# B&R Automation Studio project NAEUL004C00R13L518F00 (part 61)

#### InputRef.var - Change By Project
```iecst
(*2019-05-20*)
(**)
(*General*)
VAR
	p_eAct : REFERENCE TO eDOAction;
	p_udiMax : REFERENCE TO UDINT;
END_VAR
(**)
(*Configuration*)
VAR
	p_tyDOSettings : REFERENCE TO tyDigitalOutputSettings;
END_VAR
(**)
VAR
	p_bManual : REFERENCE TO BOOL;
	p_bSafetyRlyRst : REFERENCE TO BOOL;
	p_bTLRed : REFERENCE TO BOOL;
	p_bTLAmber : REFERENCE TO BOOL;
	p_bTLGreen : REFERENCE TO BOOL;
	p_bBuzzer : REFERENCE TO BOOL;
	p_bUSBA : REFERENCE TO BOOL;
	p_bUSBB : REFERENCE TO BOOL;
	p_bOvenInfoSigA : REFERENCE TO BOOL;
	p_bOvenInfoSigB : REFERENCE TO BOOL;
	p_bPusherExtCtrl : REFERENCE TO BOOL;
	p_bStopperUnblkCtrlA : REFERENCE TO BOOL;
	p_bStopperUnblkCtrlB : REFERENCE TO BOOL;
	p_bInletStopperRetCtrl : REFERENCE TO BOOL;
	p_eCustomerReq : REFERENCE TO eCustomer;
	p_bInletStopperExtCtrl : REFERENCE TO BOOL;
	p_bMag1SelClampCtrl : REFERENCE TO BOOL;
	p_bMag2SelClampCtrl : REFERENCE TO BOOL;
	p_bMag3SelClampCtrl : REFERENCE TO BOOL;
	p_bMag1SelUnclampCtrl : REFERENCE TO BOOL;
	p_bMag2SelUnclampCtrl : REFERENCE TO BOOL;
	p_bMag3SelUnclampCtrl : REFERENCE TO BOOL;
	p_bMag1FixedClampCtrl : REFERENCE TO BOOL;
	p_bMag1RemoteClampCtrl : REFERENCE TO BOOL;
	p_bMag2FixedClampCtrl : REFERENCE TO BOOL;
	p_bMag2RemoteClampCtrl : REFERENCE TO BOOL;
	p_bMag3FixedClampCtrl : REFERENCE TO BOOL;
	p_bMag3RemoteClampCtrl : REFERENCE TO BOOL;
	p_bInShutterOpenCtrl : REFERENCE TO BOOL;
	p_bInShutterCloseCtrl : REFERENCE TO BOOL;
	p_bOutShutterOpenCtrl : REFERENCE TO BOOL;
	p_bOutShutterCloseCtrl : REFERENCE TO BOOL;
	p_bMag1ConvMtrIn : REFERENCE TO BOOL;
	p_bMag1ConvMtrOut : REFERENCE TO BOOL;
	p_bMag2ConvMtrIn : REFERENCE TO BOOL;
	p_bMag2ConvMtrOut : REFERENCE TO BOOL;
	p_bMag3ConvMtrIn : REFERENCE TO BOOL;
	p_bMag3ConvMtrOut : REFERENCE TO BOOL;
	p_bPushConvMtrOn : REFERENCE TO BOOL;
	p_bMag1WallEngageCtrl : REFERENCE TO BOOL;
	p_bMag2WallEngageCtrl : REFERENCE TO BOOL;
	p_bMag3WallEngageCtrl : REFERENCE TO BOOL;
	p_bMag1SafetyBarRetCtrl : REFERENCE TO BOOL;
	p_bMag2SafetyBarRetCtrl : REFERENCE TO BOOL;
	p_bMag3SafetyBarRetCtrl : REFERENCE TO BOOL;
	p_bSOTMagError1 : REFERENCE TO BOOL;
	p_bSOTMagSizeLarge1 : REFERENCE TO BOOL;
	p_bSOTMagReady1 : REFERENCE TO BOOL;
	p_bSOTMagAvailable1 : REFERENCE TO BOOL;
	p_bSOTMagError2 : REFERENCE TO BOOL;
	p_bSOTMagSizeLarge2 : REFERENCE TO BOOL;
	p_bSOTMagReady2 : REFERENCE TO BOOL;
	p_bSOTMagAvailable2 : REFERENCE TO BOOL;
	p_bSOTMagError3 : REFERENCE TO BOOL;
	p_bSOTMagSizeLarge3 : REFERENCE TO BOOL;
	p_bSOTMagReady3 : REFERENCE TO BOOL;
	p_bSOTMagAvailable3 : REFERENCE TO BOOL;
	p_bSOTMagError4 : REFERENCE TO BOOL;
	p_bSOTMagSizeLarge4 : REFERENCE TO BOOL;
	p_bSOTMagReady4 : REFERENCE TO BOOL;
	p_bSOTMagAvailable4 : REFERENCE TO BOOL;
	p_bMagAWOpenLimByp1 : REFERENCE TO BOOL;
	p_bMagAWOpenLimByp2 : REFERENCE TO BOOL;
	p_bMagAWOpenLimByp3 : REFERENCE TO BOOL;
	p_bMagAWOpenLimByp4 : REFERENCE TO BOOL;
	p_bMagAWSmallLimSen1 : REFERENCE TO BOOL;
	p_bMagAWSmallLimSen2 : REFERENCE TO BOOL;
	p_bMagAWSmallLimSen3 : REFERENCE TO BOOL;
	p_bMagAWSmallLimSen4 : REFERENCE TO BOOL;
END_VAR
(**)
VAR
	p_bRequestToBring1 : REFERENCE TO BOOL;
	p_bRequestToBring2 : REFERENCE TO BOOL;
	p_bRequestToBring3 : REFERENCE TO BOOL;
	p_bRequestToBring4 : REFERENCE TO BOOL;
	p_bRequestToGet1 : REFERENCE TO BOOL;
	p_bRequestToGet2 : REFERENCE TO BOOL;
	p_bRequestToGet3 : REFERENCE TO BOOL;
	p_bRequestToGet4 : REFERENCE TO BOOL;
END_VAR
(**)
VAR
	p_bEntTopStprUnblkCtrl : REFERENCE TO BOOL;
	p_bMidTopStprUnblkCtrl : REFERENCE TO BOOL;
	p_bExtTopStprUnblkCtrl : REFERENCE TO BOOL;
	p_bMidBtmStprUnblkCtrl : REFERENCE TO BOOL;
	p_bExtBtmStprUnblkCtrl : REFERENCE TO BOOL;
	p_bEntTopStprUnblkCtrl2 : REFERENCE TO BOOL;
	p_bMidTopStprUnblkCtrl2 : REFERENCE TO BOOL;
	p_bExtTopStprUnblkCtrl2 : REFERENCE TO BOOL;
	p_bMidBtmStprUnblkCtrl2 : REFERENCE TO BOOL;
	p_bExtBtmStprUnblkCtrl2 : REFERENCE TO BOOL;
	p_bInMagConvMtrOn : REFERENCE TO BOOL;
	p_bOutMagConvMtrOn : REFERENCE TO BOOL;
	p_bInMagConv2MtrOn : REFERENCE TO BOOL;
	p_bOutMagConv2MtrOn : REFERENCE TO BOOL;
	p_bMtrPwrRly : REFERENCE TO BOOL;
END_VAR
(**)
VAR
	p_bMag1FixedClampOpenCtrl : REFERENCE TO BOOL;
	p_bMag1RemoteClampOpenCtrl : REFERENCE TO BOOL;
	p_bMag2FixedClampOpenCtrl : REFERENCE TO BOOL;
	p_bMag2RemoteClampOpenCtrl : REFERENCE TO BOOL;
	p_bMag3FixedClampOpenCtrl : REFERENCE TO BOOL;
	p_bMag3RemoteClampOpenCtrl : REFERENCE TO BOOL;
END_VAR
(**)
VAR
	p_bOutShutterOpenCtrl3 : REFERENCE TO BOOL;
	p_bOutShutterCloseCtrl3 : REFERENCE TO BOOL;
	p_bOutShutterOpenCtrl2 : REFERENCE TO BOOL;
	p_bOutShutterCloseCtrl2 : REFERENCE TO BOOL;
END_VAR
(**)
VAR
	p_bMtrPshrExt : REFERENCE TO BOOL;
	p_bMtrPshrRet : REFERENCE TO BOOL;
	p_bMtrPshrOn : REFERENCE TO BOOL;
	p_bMtrPshrBrakeRls : REFERENCE TO BOOL;
	p_bMtrPshrSpdBinBit0 : REFERENCE TO BOOL;
	p_bMtrPshrSpdBinBit1 : REFERENCE TO BOOL;
	p_bMtrPshrSpdBinBit2 : REFERENCE TO BOOL;
	p_bMtrPshrAlmRst : REFERENCE TO BOOL;
	p_bBypCurtainPBLED : REFERENCE TO BOOL;
	p_bBypCurtainSen : REFERENCE TO BOOL;
	p_bRstCurtainSen : REFERENCE TO BOOL;
END_VAR
(**)
VAR
	p_bScanTrigSig : REFERENCE TO BOOL;
	p_bMag1ExitPCB : REFERENCE TO BOOL;
	p_bMag2ExitPCB : REFERENCE TO BOOL;
	p_bMag3ExitPCB : REFERENCE TO BOOL;
END_VAR
```

### Hermes.typ - Do Not Change!!!
```iecst
(*2021-08-01*)

TYPE
	tyHermesBrdAvlDat : 	STRUCT
		a_tyXMLTableDataBrdAvl : ARRAY[0..200]OF tyXMLTableDat;
		iXMLTableDataBrdAvlTtlIdx : INT;
		bNewBrdAvl : BOOL := TRUE;
	END_STRUCT;
	tyHermesSvyParam : 	STRUCT
		tSndAlive : TIME;
		tRcvAlive : TIME;
		uiSvySvstemPort : UINT;
		iLaneID : INT;
		sMachineId : STRING[80];
		sClientAddress : STRING[15];
		uiClientPort : UINT;
		bFeatureCheckAliveResponse : BOOL;
		bFeatureConfiguration : BOOL;
		bFeatureBoardTracking : BOOL;
		bFeatureQueryWorkOrderInfo : BOOL;
		bFeatureSendWorkOrderInfo : BOOL;
		bFeatureReplyWorkOrderInfo : BOOL;
	END_STRUCT;
	tyHermesRmtParam : 	STRUCT
		uiSvrPort : UINT;
	END_STRUCT;
	tyHermesDSParam : 	STRUCT
		tSndAlive : TIME;
		tRcvAlive : TIME;
		sDownstreamInterfaceId : STRING[80]; (*The ID of the transportation interface on the downstream side*)
		uiSvrPort : UINT;
		iLaneID : INT;
		sMachineId : STRING[80] := '';
		sClientAddress : STRING[15] := '';
		uiClientPort : UINT;
		bFeatureCheckAliveResponse : BOOL;
		bFeatureBoardForecast : BOOL;
		bFeatureSendBoardInfo : BOOL;
	END_STRUCT;
	tyHermesUSParam : 	STRUCT
		tSndAlive : TIME;
		tRcvAlive : TIME;
		uiClntPort : UINT;
		iLaneID : INT;
		sMachineId : STRING[80] := '';
		sHostAddress : STRING[15] := '';
		sUpstreamInterfaceId : STRING[80]; (*The ID of the transportation interface on the upstream side*)
		uiHostPort : UINT;
		bFeatureCheckAliveResponse : BOOL;
		bFeatureBoardForecast : BOOL;
		bFeatureQueryBoardInfo : BOOL;
		bCmpTypeId : BOOL;
		bCmpParam : BOOL;
		bOverwrite : BOOL;
	END_STRUCT;
END_TYPE

(**)

TYPE
	tyHermesConfiguration : 	STRUCT
		a_tyUSParam : ARRAY[0..c_diHermesConfigMaxIdx]OF tyHermesUSParam;
		a_tyDSParam : ARRAY[0..c_diHermesConfigMaxIdx]OF tyHermesDSParam;
		tySvyParam : tyHermesSvyParam;
	END_STRUCT;
END_TYPE

(**)
(**)
(*Action*)

TYPE
	eHermesAction :
		(
		HermesActIdle,
		HermesActBGStartRun,
		HermesActBGStopRun,
		HermesActDeleteOldLog,
		HermesActCreateDir,
		HermesActWriteRetain,
		HermesActWriteRetainLane1,
		HermesActWriteRetainLane2,
		HermesActWriteRetainLane3,
		HermesActWriteRetainLane4,
		HermesActWriteRetainSendWO1,
		HermesActWriteRetainSendWO2,
		HermesActWriteRetainSendWO3,
		HermesActReadRetain,
		HermesActReadRetainLane1,
		HermesActReadRetainLane2,
		HermesActReadRetainLane3,
		HermesActReadRetainLane4,
		HermesActReadRetainSendWO1,
		HermesActReadRetainSendWO2,
		HermesActReadRetainSendWO3,
		HermesActWriteConfig,
		HermesActReadConfig
		);
END_TYPE
```

### Hermes.var - Change By Project
```iecst
(*2019-05-04*)
(**)
(*Action & State & Status*)
VAR
	p_HermesStat : UDINT;
	p_HermesStatus : UDINT;
	p_HermesStatTxt : UDINT;
END_VAR
(**)
(*Alarm*)
VAR
	p_HermesAlmData : UDINT;
END_VAR
(**)
(*Output*)
VAR
	p_HermesFileNotFound : UDINT;
	p_HermesConfiguration : UDINT;
	p_HermesConfigurationWr : UDINT;
	p_HermesUSParam1 : UDINT;
	p_HermesUSParam2 : UDINT;
	p_HermesUSParam3 : UDINT;
	p_HermesUSParam4 : UDINT;
	p_HermesDSParam1 : UDINT;
	p_HermesDSParam2 : UDINT;
	p_HermesDSParam3 : UDINT;
	p_HermesDSParam4 : UDINT;
	p_HermesSvyParam : UDINT;
	p_HermesBrdAvlDataTable1stZ : UDINT;
	p_HermesBrdAvlDataTtlIdx1stZ : UDINT;
	p_HermesBrdAvlDataNewBrdAvl1stZ : UDINT;
	p_HermesBrdAvlDataTableLastZ : UDINT;
	p_HermesBrdAvlDataTtlIdxLastZ : UDINT;
	p_HermesBrdAvlDataNewBrdAvlLastZ : UDINT;
END_VAR
```

### Program Logical/Hermes/Hermes (IEC, version 1.00.0) - 1.00.0 - NtHermes v5.00.0 , NtTCP v5.00.0 , NtMessage v5.00.0

#### Init.st - Change By Project
```iecst
(** 2021-08-01 **)
PROGRAM _INIT

	(* Always Change If Project Change *)

	//Pass Address To Global Address For External Use
	//Action, State & Status
	p_HermesStat	:= ADR(eStat);
	p_HermesStatus	:= ADR(eStatus);
	p_HermesStatTxt	:= ADR(sStatTxt);

	//Alarm
	p_HermesAlmData	:= ADR(tyAlmData);

	//Output
	p_HermesFileNotFound	        	:= ADR(bFileNotFound);
	p_HermesConfiguration	        	:= ADR(tyCurrConfiguration);
	p_HermesConfigurationWr	        	:= ADR(tyConfigurationWr);
	p_HermesUSParam1		        	:= ADR(tyCurrConfiguration.a_tyUSParam[0]); //Lane 1
	p_HermesUSParam2	        		:= ADR(tyCurrConfiguration.a_tyUSParam[1]); //Lane 2
	p_HermesUSParam3		         	:= ADR(tyCurrConfiguration.a_tyUSParam[2]); //Lane 3
	p_HermesUSParam4		        	:= ADR(tyCurrConfiguration.a_tyUSParam[3]); //Lane 4
	p_HermesDSParam1		        	:= ADR(tyCurrConfiguration.a_tyDSParam[0]); //Lane 1
	p_HermesDSParam2		        	:= ADR(tyCurrConfiguration.a_tyDSParam[1]); //Lane 2
	p_HermesDSParam3		         	:= ADR(tyCurrConfiguration.a_tyDSParam[2]); //Lane 3
	p_HermesDSParam4		        	:= ADR(tyCurrConfiguration.a_tyDSParam[3]); //Lane 4
	p_HermesSvyParam		        	:= ADR(tyCurrConfiguration.tySvyParam);
	p_HermesBrdAvlDataTable1stZ		    := ADR(a_tyHermesBrdAvlData[1].a_tyXMLTableDataBrdAvl); //Lane 1 First Zone Data, for B.F
	p_HermesBrdAvlDataTtlIdx1stZ    	:= ADR(a_tyHermesBrdAvlData[1].iXMLTableDataBrdAvlTtlIdx);  //Lane 1 First Zone Data, for B.F
	p_HermesBrdAvlDataNewBrdAvl1stZ	    := ADR(a_tyHermesBrdAvlData[1].bNewBrdAvl);  //Lane 1 First Zone Data, for B.F
	p_HermesBrdAvlDataTableLastZ		:= ADR(a_tyHermesBrdAvlData[1].a_tyXMLTableDataBrdAvl); //Lane 1 Last Zone Data,for B.A, adjust array no. accordingly
	p_HermesBrdAvlDataTtlIdxLastZ	    := ADR(a_tyHermesBrdAvlData[1].iXMLTableDataBrdAvlTtlIdx); //Lane 1 Last Zone Data,for B.A, adjust array no. accordingly
	p_HermesBrdAvlDataNewBrdAvlLastZ	:= ADR(a_tyHermesBrdAvlData[1].bNewBrdAvl); //Lane 1 Last Zone Data,for B.A, adjust array no. accordingly

	(* Always Change If Project Change *)
END_PROGRAM
```

#### Act_InitGlobal.st - Change By Project
```iecst
(** 2021-08-01 **)
ACTION Act_InitGlobal:

	(* Always Change If Project Change *)

	//Pass Data To Link
	p_bLinkStartupRun ACCESS p_StartupRun;

	pa_tyLinkXMLTableDataBrdAvl1 ACCESS p_USHermesATableDataBrdAvl; //lane 1 B.A
	p_iLinkXMLTableDataBrdAvlTtlIdx1 ACCESS p_USHermesATableDataBrdAvlTtlIdx; //lane 1 B.A
//	pa_tyLinkXMLTableDataBrdAvl2 ACCESS p_USHermesTableDataBrdAvl2; //lane 2 B.A
//	p_iLinkXMLTableDataBrdAvlTtlIdx2 ACCESS p_USHermesTableDataBrdAvlTtlIdx2; //lane 2 B.A
//	pa_tyLinkXMLTableDataBrdAvl3 ACCESS p_USHermesTableDataBrdAvl3; //lane 3 B.A
//	p_iLinkXMLTableDataBrdAvlTtlIdx3 ACCESS p_USHermesTableDataBrdAvlTtlIdx3; //lane 3 B.A
//	pa_tyLinkXMLTableDataBrdAvl4 ACCESS p_USHermesTableDataBrdAvl4; //lane 4 B.A
//	p_iLinkXMLTableDataBrdAvlTtlIdx4 ACCESS p_USHermesTableDataBrdAvlTtlIdx4; //lane 4 B.A
	p_eLinkTravLifULPosGo ACCESS p_OpsTravLifULPosGo;
	p_bLinkOpsTravLifULInitDone ACCESS p_OpsTravLifULInitDone; //p_OpsInitConvStepInitDone;
//	p_bLinkOpsInitGConv1MidHvBrd ACCESS p_OpsInitConvMidHvBrd;
	p_bLinkOpsTravLifULEntBrd ACCESS p_OpsTravLifULEntBrd;
	p_bLinkOpsTravLifULExitBrd ACCESS p_OpsTravLifULExitBrd;
	p_bLinkConvHvBrd ACCESS p_PshrConvHvBrd; //p_ConvHvBrd

	p_bLinkUSHermesTransporting ACCESS p_USHermesATransporting;
	p_bLinkUSSMEMATransporting ACCESS p_USSMEMAATransporting;
//	p_bLinkOpsGConv1StepEntBrd ACCESS p_OpsTravLifULEntBrd;// p_OpsConvStepEntBrd;
//	p_bLinkOpsInitGConv2StepInitDone ACCESS p_OpsInitGConv2StepInitDone;  //Zone2
//	p_bLinkOpsInitGConv2MidHvBrd ACCESS p_OpsInitGConv2MidHvBrd;  //Zone2
//	p_bLinkOpsInitGConv2EndHvBrd ACCESS p_OpsInitGConv2EndHvBrd;  //Zone2
//	p_bLinkOpsGConv2HvBrd ACCESS p_OpsGConv2HvBrd;  //Zone2
//	p_bLinkOpsGConv2StepEntBrd ACCESS p_OpsGConv2StepEntBrd;  //Zone2
//	p_bLinkUSSMEMA2Transporting ACCESS p_USSMEMA2Transporting;  //Zone2

	//Pass Data To Internal Use
	p_udiRstErr ACCESS p_RstErrReset;
	p_bPrep ACCESS p_NtParamHermesPrep;
	pa_tyUSParam ACCESS p_UIHermesUSParamWr; //HMI US Configure from UI
	//pa_tyDSParam ACCESS p_UIHermesDSParamWr; //HMI DS Configure from UI
	p_tySvyParam ACCESS p_UIHermesSvyParamWr; //HMI Svy Configure from UI
	p_tyRmtSetConfiguration ACCESS p_RmtHermesSetConfiguration; //US,DS SetConfigure from RmtHermes
	p_tySvySetConfiguration ACCESS p_SvyHermesSetConfiguration; //US,DS SetConfigure from SvyHermes
	p_bRmtPrep ACCESS p_NtParamHermesRmtPrep;
	p_bRmtEn ACCESS p_McParamHermesRmtEn;
	p_bSvyPrep ACCESS p_NtParamHermesSvyPrep;
	p_bSvyEn ACCESS p_McParamHermesSvyEn;
	p_sRetainFileName1 ACCESS p_NtParamHermesRetainFileNm; //lane 1
//	p_sRetainFileName2 ACCESS p_NtParamHermesRetainFileNm2; //lane 2, rename to HermesL2.dat
//	p_sRetainFileName3 ACCESS p_NtParamHermesRetainFileNm3; //lane 3, rename to HermesL3.dat
//	p_sRetainFileName4 ACCESS p_NtParamHermesRetainFileNm4; //lane 4, rename to HermesL4.dat
	p_sConfigFileName ACCESS p_NtParamHermesConfigFileNm;
	p_sProgNm ACCESS p_NtParamHermesProgNm;
	p_bNtSettingsLoadDone ACCESS p_StartupNtSettingsLoadDone;
	p_bRmtHermesWriteConfig ACCESS p_RmtHermesWriteConfig;
	p_bSvyHermesWriteConfig ACCESS p_SvyHermesWriteConfig;
	p_bUISaveHMIConfigure ACCESS p_UISaveHMIConfigure;
	p_bUISaveHMISvyConfig ACCESS p_UISaveHMISvyConfig;
	p_sMcId ACCESS p_McParamMcNm;

	p_bRmtFoundIndexUS1 ACCESS p_RmtHermesFoundIndexUS1;
	p_bRmtFoundIndexUS2 ACCESS p_RmtHermesFoundIndexUS2;
	p_bRmtFoundIndexUS3 ACCESS p_RmtHermesFoundIndexUS3;
	p_bRmtFoundIndexUS4 ACCESS p_RmtHermesFoundIndexUS4;
	p_bRmtFoundIndexDS1 ACCESS p_RmtHermesFoundIndexDS1;
	p_bRmtFoundIndexDS2 ACCESS p_RmtHermesFoundIndexDS2;
	p_bRmtFoundIndexDS3 ACCESS p_RmtHermesFoundIndexDS3;
	p_bRmtFoundIndexDS4 ACCESS p_RmtHermesFoundIndexDS4;
	p_udiRmtIndexUS1 ACCESS p_RmtHermesIndexUS1;
	p_udiRmtIndexUS2 ACCESS p_RmtHermesIndexUS2;
	p_udiRmtIndexUS3 ACCESS p_RmtHermesIndexUS3;
	p_udiRmtIndexUS4 ACCESS p_RmtHermesIndexUS4;
	p_udiRmtIndexDS1 ACCESS p_RmtHermesIndexDS1;
	p_udiRmtIndexDS2 ACCESS p_RmtHermesIndexDS2;
	p_udiRmtIndexDS3 ACCESS p_RmtHermesIndexDS3;
	p_udiRmtIndexDS4 ACCESS p_RmtHermesIndexDS4;

	p_bSvyFoundIndexUS1 ACCESS p_SvyHermesFoundIndexUS1;
	p_bSvyFoundIndexUS2 ACCESS p_SvyHermesFoundIndexUS2;
	p_bSvyFoundIndexUS3 ACCESS p_SvyHermesFoundIndexUS3;
	p_bSvyFoundIndexUS4 ACCESS p_SvyHermesFoundIndexUS4;
	p_bSvyFoundIndexDS1 ACCESS p_SvyHermesFoundIndexDS1;
	p_bSvyFoundIndexDS2 ACCESS p_SvyHermesFoundIndexDS2;
	p_bSvyFoundIndexDS3 ACCESS p_SvyHermesFoundIndexDS3;
	p_bSvyFoundIndexDS4 ACCESS p_SvyHermesFoundIndexDS4;
	p_udiSvyIndexUS1 ACCESS p_SvyHermesIndexUS1;
	p_udiSvyIndexUS2 ACCESS p_SvyHermesIndexUS2;
	p_udiSvyIndexUS3 ACCESS p_SvyHermesIndexUS3;
	p_udiSvyIndexUS4 ACCESS p_SvyHermesIndexUS4;
	p_udiSvyIndexDS1 ACCESS p_SvyHermesIndexDS1;
	p_udiSvyIndexDS2 ACCESS p_SvyHermesIndexDS2;
	p_udiSvyIndexDS3 ACCESS p_SvyHermesIndexDS3;
	p_udiSvyIndexDS4 ACCESS p_SvyHermesIndexDS4;

	p_eLinkMcParamUSACommMod ACCESS p_McParamUSCommAMod;
	p_eLinkMcParamUSBCommMod ACCESS p_McParamUSCommBMod;

	p_bLinkDIRightSen ACCESS p_DIConvRgtSen;
	p_bLinkDIClrSen ACCESS p_DIConvClrSen;

	(* Always Change If Project Change *)
END_ACTION
```

#### InputRef_Link.var - Change By Project
```iecst
(*2021-08-01*)
(**)
VAR
	p_bLinkStartupRun : REFERENCE TO BOOL;
END_VAR
(**)
VAR
	p_eLinkMcParamUSACommMod : REFERENCE TO eMcSetCommMod;
	p_eLinkMcParamUSBCommMod : REFERENCE TO eMcSetCommMod;
	pa_tyLinkXMLTableDataBrdAvl1 : REFERENCE TO ARRAY[0..200] OF tyXMLTableDat;
	p_iLinkXMLTableDataBrdAvlTtlIdx1 : REFERENCE TO INT;
	pa_tyLinkXMLTableDataBrdAvl2 : REFERENCE TO ARRAY[0..200] OF tyXMLTableDat;
	p_iLinkXMLTableDataBrdAvlTtlIdx2 : REFERENCE TO INT;
	pa_tyLinkXMLTableDataBrdAvl3 : REFERENCE TO ARRAY[0..200] OF tyXMLTableDat;
	p_iLinkXMLTableDataBrdAvlTtlIdx3 : REFERENCE TO INT;
	pa_tyLinkXMLTableDataBrdAvl4 : REFERENCE TO ARRAY[0..200] OF tyXMLTableDat;
	p_iLinkXMLTableDataBrdAvlTtlIdx4 : REFERENCE TO INT;
END_VAR
(**)
VAR
	tyHermesBrdAvlData : tyHermesBrdAvlDat;
	a_tyHermesBrdAvlData : ARRAY[1..200] OF tyHermesBrdAvlDat; (*Cater Up to 6 Zones*)
END_VAR
(**)
(*Zone 1*)
VAR
	p_eLinkTravLifULPosGo : REFERENCE TO eTravLifULPos;
	p_bLinkOpsTravLifULInitDone : REFERENCE TO BOOL;
	p_bLinkOpsTravLifULEntBrd : REFERENCE TO BOOL;
	p_bLinkOpsTravLifULExitBrd : REFERENCE TO BOOL;
	p_bLinkConvHvBrd : REFERENCE TO BOOL;
	p_bLinkDIRightSen : REFERENCE TO BOOL;
	p_bLinkDIClrSen : REFERENCE TO BOOL;
	p_bLinkOpsInitGConv1MidHvBrd : REFERENCE TO BOOL;
	p_bLinkOpsInitGConv1EndHvBrd : REFERENCE TO BOOL;
	p_bLinkOpsGConv1StepEntBrd : REFERENCE TO BOOL;
	p_bLinkUSHermesTransporting : REFERENCE TO BOOL;
	p_bLinkUSSMEMATransporting : REFERENCE TO BOOL;
END_VAR
(**)
(*Zone 2*)
VAR
	p_bLinkOpsInitGConv2StepInitDone : REFERENCE TO BOOL;
	p_bLinkOpsInitGConv2MidHvBrd : REFERENCE TO BOOL;
	p_bLinkOpsInitGConv2EndHvBrd : REFERENCE TO BOOL;
	p_bLinkOpsGConv2HvBrd : REFERENCE TO BOOL;
	p_bLinkOpsGConv2StepEntBrd : REFERENCE TO BOOL;
	p_bLinkUSSMEMA2Transporting : REFERENCE TO BOOL;
END_VAR
(**)
```

#### Act_LinkAction.st - Change By Project
```iecst
(** 2021-08-01 **)
ACTION Act_LinkAction:

	IF p_bLinkStartupRun = TRUE THEN
		p_eAct ACCESS p_StartupHermesAct;
	ELSIF p_bSvyHermesWriteConfig THEN //Changed
		p_eAct ACCESS p_SvyHermesAct;
	ELSIF p_bRmtHermesWriteConfig THEN
		p_eAct ACCESS p_RmtHermesAct;
	ELSIF p_bUISaveHMIConfigure OR p_bUISaveHMISvyConfig THEN //Change
		p_eAct ACCESS p_UIHermesAct;
	END_IF

END_ACTION
```

#### Act_Link.st - Change By Project
```iecst
(** 2019-05-04 **)
ACTION Act_Link:

	//If not two lane operating at same time no need Lane
	p_udiRetainDataAddr1	:= ADR(a_tyHermesBrdAvlData);
	p_udiRetainDataLen1  	:= SIZEOF(a_tyHermesBrdAvlData);

	IF p_bLinkStartupRun = FALSE THEN

		//Passing Board Available Memory
		//Init Board
		IF EDGEPOS(p_bLinkOpsTravLifULInitDone = TRUE) THEN

			IF p_bLinkConvHvBrd = FALSE THEN
				a_tyHermesBrdAvlData[1].bNewBrdAvl	:= TRUE;

				bHermesWriteRetainLane1	:= TRUE;
			END_IF

		END_IF

		//Enter Board - US1
		IF p_eLinkTravLifULPosGo = TravLifULPosUS1 AND p_bLinkOpsTravLifULEntBrd = TRUE AND EDGEPOS(p_bLinkConvHvBrd = TRUE) THEN

			IF p_eLinkMcParamUSACommMod = McSetCommModHermes THEN

				a_tyHermesBrdAvlData[1].a_tyXMLTableDataBrdAvl		:= pa_tyLinkXMLTableDataBrdAvl1;
				a_tyHermesBrdAvlData[1].iXMLTableDataBrdAvlTtlIdx	:= p_iLinkXMLTableDataBrdAvlTtlIdx1;
				a_tyHermesBrdAvlData[1].bNewBrdAvl					:= FALSE;

				bHermesWriteRetainLane1	:= TRUE;

			ELSE

				a_tyHermesBrdAvlData[1].bNewBrdAvl	:= TRUE;

				bHermesWriteRetainLane1	:= TRUE;

			END_IF

		END_IF

		//Enter Board - US2
		IF p_eLinkTravLifULPosGo = TravLifULPosUS2 AND p_bLinkOpsTravLifULEntBrd = TRUE AND EDGEPOS(p_bLinkConvHvBrd = TRUE) THEN

			IF p_eLinkMcParamUSBCommMod = McSetCommModHermes THEN

				a_tyHermesBrdAvlData[1].a_tyXMLTableDataBrdAvl		:= pa_tyLinkXMLTableDataBrdAvl2;
				a_tyHermesBrdAvlData[1].iXMLTableDataBrdAvlTtlIdx	:= p_iLinkXMLTableDataBrdAvlTtlIdx2;
				a_tyHermesBrdAvlData[1].bNewBrdAvl					:= FALSE;

				bHermesWriteRetain	:= TRUE;

			ELSE

				a_tyHermesBrdAvlData[1].bNewBrdAvl	:= TRUE;

				bHermesWriteRetain	:= TRUE;

			END_IF

		END_IF

		//Exit Board
		IF p_bLinkOpsTravLifULExitBrd = TRUE AND EDGEPOS(p_bLinkConvHvBrd = FALSE  AND EDGENEG(p_bLinkDIRightSen OR p_bLinkDIClrSen )) THEN
			a_tyHermesBrdAvlData[1].bNewBrdAvl	:= TRUE;
			bHermesWriteRetainLane1	:= TRUE;
		END_IF

		//Write Hermes Retain Data
		IF bHermesWriteRetainLane1 = TRUE THEN
			p_eAct	:= HermesActWriteRetainLane1;

			IF (eStat = HermesActWriteRetainLane1) AND (eStatus = Done) THEN
				p_eAct				:= HermesActIdle;
				bHermesWriteRetainLane1	:= FALSE;
			END_IF
		END_IF

	END_IF

END_ACTION
```

#### Cyclic.st - Do Not Change!!!
```iecst
(** 2021-08-01 **)
PROGRAM _CYCLIC

	IF bInitDone = FALSE THEN
		bInitDone	:= TRUE;

		Act_InitLocal;
		Act_InitGlobal;

	ELSIF bInitialDone = FALSE THEN
		IF p_bNtSettingsLoadDone = TRUE THEN
			bInitialDone	:= TRUE;

			Act_Initial;
		END_IF

	ELSE

		Act_RstErr;
		Act_LinkAction;
		Act_Action;
		Act_LinkEn;

		IF (p_bPrep = TRUE) AND (p_bEn = TRUE) AND (p_bDis = FALSE) THEN
			Act_Link;
			Act_Background;
			Act_Main;

		ELSE
			IF eStat <> HermesActIdle THEN
				eStatus	:= Done;
			ELSE
				eStatus	:= Idle;
			END_IF
		END_IF

		Act_Alarm;

	END_IF

END_PROGRAM
```

#### Act_Initial.st - Do Not Change!!!
```iecst
(** 2021-08-01 **)
ACTION Act_Initial:

	//Initial
	sStatTxt	:= a_sStatText[eStat];

	fbDirCreate1.sDevice	:= 'F';
	fbDirCreate1.sDirName	:= 'User';
	fbDirCreate1(bEn := FALSE);

	fbDirCreate2.sDevice	:= 'User';
	fbDirCreate2.sDirName	:= 'Retain';
	fbDirCreate2(bEn := FALSE);

	fbDirCreate3.sDevice	:= 'User';
	fbDirCreate3.sDirName	:= 'Log';
	fbDirCreate3(bEn := FALSE);

	fbDirCreate4.sDevice	:= 'User';
	fbDirCreate4.sDirName	:= 'MachineParameter';
	fbDirCreate4(bEn := FALSE);

	fbFileRead1.sDevice			:= 'McParam';
	fbFileRead1.sFile			:= p_sConfigFileName;
	fbFileRead1.udiOffset		:= 0;
	fbFileRead1.p_Dest			:= ADR(tyCurrConfiguration);
	fbFileRead1.udiLen			:= SIZEOF(tyCurrConfiguration);
	fbFileRead1(bEn := FALSE);

	fbFileWrite1.sDevice		:= 'McParam';
	fbFileWrite1.sFile			:= p_sConfigFileName;
	fbFileWrite1.udiOffset		:= 0;
	fbFileWrite1.p_Src			:= ADR(tyConfigurationWr);
	fbFileWrite1.udiLen			:= SIZEOF(tyConfigurationWr);
	fbFileWrite1.udiOption		:= 0;
	fbFileWrite1(bEn := FALSE);

	fbFileRead2.sDevice			:= 'Retain';
	fbFileRead2.sFile			:= p_sRetainFileName1;
	fbFileRead2.udiOffset		:= 0;
	fbFileRead2(bEn := FALSE);

	fbFileWrite2.sDevice		:= 'Retain';
	fbFileWrite2.sFile			:= p_sRetainFileName1;
	fbFileWrite2.udiOffset		:= 0;
	fbFileWrite2.udiOption		:= 0;
	fbFileWrite2(bEn := FALSE);

	fbFileRead3.sDevice			:= 'Retain';
	fbFileRead3.sFile			:= p_sRetainFileName2;
	fbFileRead3.udiOffset		:= 0;
	fbFileRead3(bEn := FALSE);

	fbFileWrite3.sDevice		:= 'Retain';
	fbFileWrite3.sFile			:= p_sRetainFileName2;
	fbFileWrite3.udiOffset		:= 0;
	fbFileWrite3.udiOption		:= 0;
	fbFileWrite3(bEn := FALSE);

	fbFileRead4.sDevice			:= 'Retain';
	fbFileRead4.sFile			:= p_sRetainFileName3;
	fbFileRead4.udiOffset		:= 0;
	fbFileRead4(bEn := FALSE);

	fbFileWrite4.sDevice		:= 'Retain';
	fbFileWrite4.sFile			:= p_sRetainFileName3;
	fbFileWrite4.udiOffset		:= 0;
	fbFileWrite4.udiOption		:= 0;
	fbFileWrite4(bEn := FALSE);

	fbFileRead5.sDevice			:= 'Retain';
	fbFileRead5.sFile			:= p_sRetainFileName4;
	fbFileRead5.udiOffset		:= 0;
	fbFileRead5(bEn := FALSE);

	fbFileWrite5.sDevice		:= 'Retain';
	fbFileWrite5.sFile			:= p_sRetainFileName4;
	fbFileWrite5.udiOffset		:= 0;
	fbFileWrite5.udiOption		:= 0;
	fbFileWrite5(bEn := FALSE);

END_ACTION
```

#### Act_InitLocal.st - Do Not Change!!!
```iecst
(** 2021-08-01 **)
ACTION Act_InitLocal:

	//Input Reference Link To Local Variable
	p_eAct ACCESS ADR(eAct);
	p_udiRstErr ACCESS ADR(udiRstErr);
	p_bPrep ACCESS ADR(bPrep);
	p_bEn ACCESS ADR(bEn);
	p_bDis ACCESS ADR(bDis);
	pa_tyUSParam ACCESS ADR(a_tyUSParam);
	pa_tyDSParam ACCESS ADR(a_tyDSParam);
	p_tyRmtParam ACCESS ADR(tyRmtParam);
	p_tySvyParam ACCESS ADR(tySvyParam);
	p_tyRmtSetConfiguration ACCESS ADR(tyRmtSetConfiguration);
	p_tySvySetConfiguration ACCESS ADR(tySvySetConfiguration);
	p_bRmtPrep ACCESS ADR(bRmtPrep);
	p_bRmtEn ACCESS ADR(bRmtEn);
	p_bSvyPrep ACCESS ADR(bSvyPrep);
	p_bSvyEn ACCESS ADR(bSvyEn);
	p_sRetainFileName1 ACCESS ADR(sRetainFileName1);
	p_sRetainFileName2 ACCESS ADR(sRetainFileName2);
	p_sRetainFileName3 ACCESS ADR(sRetainFileName3);
	p_sRetainFileName4 ACCESS ADR(sRetainFileName4);
	p_udiRetainDataAddr1 ACCESS ADR(udiRetainDataAddr1);
	p_udiRetainDataLen1 ACCESS ADR(udiRetainDataLen1);
	p_udiRetainDataAddr2 ACCESS ADR(udiRetainDataAddr2);
	p_udiRetainDataLen2 ACCESS ADR(udiRetainDataLen2);
	p_udiRetainDataAddr3 ACCESS ADR(udiRetainDataAddr3);
	p_udiRetainDataLen3 ACCESS ADR(udiRetainDataLen3);
	p_udiRetainDataAddr4 ACCESS ADR(udiRetainDataAddr4);
	p_udiRetainDataLen4 ACCESS ADR(udiRetainDataLen4);
	p_sConfigFileName ACCESS ADR(sConfigFileName);
	p_sProgNm ACCESS ADR(sProgNm);
	p_bNtSettingsLoadDone ACCESS ADR(bNtSettingsLoadDone);
	p_bRmtHermesWriteConfig ACCESS ADR(bRmtHermesWriteConfig);
	p_bSvyHermesWriteConfig ACCESS ADR(bSvyHermesWriteConfig);
	p_bUISaveHMIConfigure ACCESS ADR(bUISaveHMIConfigure);
	p_bUISaveHMISvyConfig ACCESS ADR(bUISaveHMISvyConfig);
	p_sMcId ACCESS ADR(sMcId);

	p_bRmtFoundIndexUS1 ACCESS ADR(bRmtFoundIndexUS1);
	p_bRmtFoundIndexUS2 ACCESS ADR(bRmtFoundIndexUS2);
	p_bRmtFoundIndexUS3 ACCESS ADR(bRmtFoundIndexUS3);
	p_bRmtFoundIndexUS4 ACCESS ADR(bRmtFoundIndexUS4);
	p_bRmtFoundIndexDS1 ACCESS ADR(bRmtFoundIndexDS1);
	p_bRmtFoundIndexDS2 ACCESS ADR(bRmtFoundIndexDS2);
	p_bRmtFoundIndexDS3 ACCESS ADR(bRmtFoundIndexDS3);
	p_bRmtFoundIndexDS4 ACCESS ADR(bRmtFoundIndexDS4);
	p_udiRmtIndexUS1 ACCESS ADR(udiRmtIndexUS1);
	p_udiRmtIndexUS2 ACCESS ADR(udiRmtIndexUS2);
	p_udiRmtIndexUS3 ACCESS ADR(udiRmtIndexUS3);
	p_udiRmtIndexUS4 ACCESS ADR(udiRmtIndexUS4);
	p_udiRmtIndexDS1 ACCESS ADR(udiRmtIndexDS1);
	p_udiRmtIndexDS2 ACCESS ADR(udiRmtIndexDS2);
	p_udiRmtIndexDS3 ACCESS ADR(udiRmtIndexDS3);
	p_udiRmtIndexDS4 ACCESS ADR(udiRmtIndexDS4);

	p_bSvyFoundIndexUS1 ACCESS ADR(bSvyFoundIndexUS1);
	p_bSvyFoundIndexUS2 ACCESS ADR(bSvyFoundIndexUS2);
	p_bSvyFoundIndexUS3 ACCESS ADR(bSvyFoundIndexUS3);
	p_bSvyFoundIndexUS4 ACCESS ADR(bSvyFoundIndexUS4);
	p_bSvyFoundIndexDS1 ACCESS ADR(bSvyFoundIndexDS1);
	p_bSvyFoundIndexDS2 ACCESS ADR(bSvyFoundIndexDS2);
	p_bSvyFoundIndexDS3 ACCESS ADR(bSvyFoundIndexDS3);
	p_bSvyFoundIndexDS4 ACCESS ADR(bSvyFoundIndexDS4);
	p_udiSvyIndexUS1 ACCESS ADR(udiSvyIndexUS1);
	p_udiSvyIndexUS2 ACCESS ADR(udiSvyIndexUS2);
	p_udiSvyIndexUS3 ACCESS ADR(udiSvyIndexUS3);
	p_udiSvyIndexUS4 ACCESS ADR(udiSvyIndexUS4);
	p_udiSvyIndexDS1 ACCESS ADR(udiSvyIndexDS1);
	p_udiSvyIndexDS2 ACCESS ADR(udiSvyIndexDS2);
	p_udiSvyIndexDS3 ACCESS ADR(udiSvyIndexDS3);
	p_udiSvyIndexDS4 ACCESS ADR(udiSvyIndexDS4);

	//Changed
//	p_bSvyPrep ACCESS ADR(bVoid);
//	p_bSvyEn ACCESS ADR(bVoid);
	p_bSvyHermesWriteConfig ACCESS ADR(bSvyHermesWriteConfig);
END_ACTION
```

#### Act_Action.st - Do Not Change!!!
```iecst
(** 2021-08-01 **)
ACTION Act_Action:

	//Reset Error
	IF (eStatus = Error) AND bRstErr THEN
		p_eAct	:= HermesActIdle;
		eStat	:= HermesActIdle;
	END_IF

	//Set p_eAct
	IF eStatus = Idle (*OR eStatus = Busy*) OR eStatus = Done THEN
		eStat	:= p_eAct;
	END_IF

END_ACTION
```

#### Act_Background.st - Do Not Change!!!
```iecst
(** 2021-08-01 **)
ACTION Act_Background:

	//Update Configuration
		//Changed
	IF p_bSvyPrep = TRUE AND p_bSvyEn = TRUE AND p_bSvyHermesWriteConfig THEN

		IF p_bSvyFoundIndexUS1 THEN
			tyConfigurationWr.a_tyUSParam[0].iLaneID		            := p_tySvySetConfiguration.tyData.a_tyUpstreamConfigurations[p_udiSvyIndexUS1].iUpstreamLaneId;
			tyConfigurationWr.a_tyUSParam[0].sHostAddress           	:= p_tySvySetConfiguration.tyData.a_tyUpstreamConfigurations[p_udiSvyIndexUS1].sHostAddress;
			tyConfigurationWr.a_tyUSParam[0].uiHostPort	                := p_tySvySetConfiguration.tyData.a_tyUpstreamConfigurations[p_udiSvyIndexUS1].uiPort;
			tyConfigurationWr.a_tyUSParam[0].sUpstreamInterfaceId   	:= p_tySvySetConfiguration.tyData.a_tyUpstreamConfigurations[p_udiSvyIndexUS1].sUpstreamInterfaceId;
		END_IF

		IF p_bSvyFoundIndexUS2 THEN
			tyConfigurationWr.a_tyUSParam[1].iLaneID		            := p_tySvySetConfiguration.tyData.a_tyUpstreamConfigurations[p_udiSvyIndexUS2].iUpstreamLaneId;
			tyConfigurationWr.a_tyUSParam[1].sHostAddress           	:= p_tySvySetConfiguration.tyData.a_tyUpstreamConfigurations[p_udiSvyIndexUS2].sHostAddress;
			tyConfigurationWr.a_tyUSParam[1].uiHostPort	                := p_tySvySetConfiguration.tyData.a_tyUpstreamConfigurations[p_udiSvyIndexUS2].uiPort;
			tyConfigurationWr.a_tyUSParam[1].sUpstreamInterfaceId   	:= p_tySvySetConfiguration.tyData.a_tyUpstreamConfigurations[p_udiSvyIndexUS2].sUpstreamInterfaceId;
		END_IF

		IF p_bSvyFoundIndexUS3 THEN
			tyConfigurationWr.a_tyUSParam[2].iLaneID		            := p_tySvySetConfiguration.tyData.a_tyUpstreamConfigurations[p_udiSvyIndexUS3].iUpstreamLaneId;
			tyConfigurationWr.a_tyUSParam[2].sHostAddress           	:= p_tySvySetConfiguration.tyData.a_tyUpstreamConfigurations[p_udiSvyIndexUS3].sHostAddress;
			tyConfigurationWr.a_tyUSParam[2].uiHostPort	                := p_tySvySetConfiguration.tyData.a_tyUpstreamConfigurations[p_udiSvyIndexUS3].uiPort;
			tyConfigurationWr.a_tyUSParam[2].sUpstreamInterfaceId   	:= p_tySvySetConfiguration.tyData.a_tyUpstreamConfigurations[p_udiSvyIndexUS3].sUpstreamInterfaceId;
		END_IF

		IF p_bSvyFoundIndexUS4 THEN
			tyConfigurationWr.a_tyUSParam[3].iLaneID		            := p_tySvySetConfiguration.tyData.a_tyUpstreamConfigurations[p_udiSvyIndexUS4].iUpstreamLaneId;
			tyConfigurationWr.a_tyUSParam[3].sHostAddress           	:= p_tySvySetConfiguration.tyData.a_tyUpstreamConfigurations[p_udiSvyIndexUS4].sHostAddress;
			tyConfigurationWr.a_tyUSParam[3].uiHostPort	                := p_tySvySetConfiguration.tyData.a_tyUpstreamConfigurations[p_udiSvyIndexUS4].uiPort;
			tyConfigurationWr.a_tyUSParam[3].sUpstreamInterfaceId   	:= p_tySvySetConfiguration.tyData.a_tyUpstreamConfigurations[p_udiSvyIndexUS4].sUpstreamInterfaceId;
		END_IF

		IF p_bSvyFoundIndexDS1 THEN
			tyConfigurationWr.a_tyDSParam[0].iLaneID	            	:= p_tySvySetConfiguration.tyData.a_tyDownstreamConfigurations[p_udiSvyIndexDS1].iDownstreamLaneId;
			tyConfigurationWr.a_tyDSParam[0].uiSvrPort               	:= p_tySvySetConfiguration.tyData.a_tyDownstreamConfigurations[p_udiSvyIndexDS1].uiPort;
			tyConfigurationWr.a_tyDSParam[0].sDownstreamInterfaceId  	:= p_tySvySetConfiguration.tyData.a_tyDownstreamConfigurations[p_udiSvyIndexDS1].sDownstreamInterfaceId;
		END_IF

		IF p_bSvyFoundIndexDS2 THEN
			tyConfigurationWr.a_tyDSParam[1].iLaneID	            	:= p_tySvySetConfiguration.tyData.a_tyDownstreamConfigurations[p_udiSvyIndexDS2].iDownstreamLaneId;
			tyConfigurationWr.a_tyDSParam[1].uiSvrPort               	:= p_tySvySetConfiguration.tyData.a_tyDownstreamConfigurations[p_udiSvyIndexDS2].uiPort;
			tyConfigurationWr.a_tyDSParam[1].sDownstreamInterfaceId  	:= p_tySvySetConfiguration.tyData.a_tyDownstreamConfigurations[p_udiSvyIndexDS2].sDownstreamInterfaceId;
		END_IF

		IF p_bSvyFoundIndexDS3 THEN
			tyConfigurationWr.a_tyDSParam[2].iLaneID	            	:= p_tySvySetConfiguration.tyData.a_tyDownstreamConfigurations[p_udiSvyIndexDS3].iDownstreamLaneId;
			tyConfigurationWr.a_tyDSParam[2].uiSvrPort               	:= p_tySvySetConfiguration.tyData.a_tyDownstreamConfigurations[p_udiSvyIndexDS3].uiPort;
			tyConfigurationWr.a_tyDSParam[2].sDownstreamInterfaceId  	:= p_tySvySetConfiguration.tyData.a_tyDownstreamConfigurations[p_udiSvyIndexDS3].sDownstreamInterfaceId;
		END_IF

		IF p_bSvyFoundIndexDS4 THEN
			tyConfigurationWr.a_tyDSParam[3].iLaneID	            	:= p_tySvySetConfiguration.tyData.a_tyDownstreamConfigurations[p_udiSvyIndexDS4].iDownstreamLaneId;
			tyConfigurationWr.a_tyDSParam[3].uiSvrPort               	:= p_tySvySetConfiguration.tyData.a_tyDownstreamConfigurations[p_udiSvyIndexDS4].uiPort;
			tyConfigurationWr.a_tyDSParam[3].sDownstreamInterfaceId  	:= p_tySvySetConfiguration.tyData.a_tyDownstreamConfigurations[p_udiSvyIndexDS4].sDownstreamInterfaceId;
		END_IF

		IF p_tySvySetConfiguration.tyAvl.bMachineId = TRUE THEN

			tyConfigurationWr.a_tyUSParam[0].sMachineId		:= p_tySvySetConfiguration.tyData.sMachineId;
			tyConfigurationWr.a_tyDSParam[0].sMachineId		:= p_tySvySetConfiguration.tyData.sMachineId;
			tyConfigurationWr.tySvyParam.sMachineId		    := p_tySvySetConfiguration.tyData.sMachineId;

		END_IF

		IF p_tySvySetConfiguration.tyAvl.bSupervisorySystemPort = TRUE THEN

			tyConfigurationWr.tySvyParam.uiSvySvstemPort	:= p_tySvySetConfiguration.tyData.uiSupervisorySystemPort;

		END_IF

	ELSIF p_bRmtPrep = TRUE AND p_bRmtEn = TRUE AND p_bRmtHermesWriteConfig THEN

		IF p_bRmtFoundIndexUS1 THEN
			tyConfigurationWr.a_tyUSParam[0].iLaneID		            := p_tyRmtSetConfiguration.tyData.a_tyUpstreamConfigurations[p_udiRmtIndexUS1].iUpstreamLaneId;
			tyConfigurationWr.a_tyUSParam[0].sHostAddress           	:= p_tyRmtSetConfiguration.tyData.a_tyUpstreamConfigurations[p_udiRmtIndexUS1].sHostAddress;
			tyConfigurationWr.a_tyUSParam[0].uiHostPort	                := p_tyRmtSetConfiguration.tyData.a_tyUpstreamConfigurations[p_udiRmtIndexUS1].uiPort;
			tyConfigurationWr.a_tyUSParam[0].sUpstreamInterfaceId   	:= p_tyRmtSetConfiguration.tyData.a_tyUpstreamConfigurations[p_udiRmtIndexUS1].sUpstreamInterfaceId;
		END_IF

		IF p_bRmtFoundIndexUS2 THEN
			tyConfigurationWr.a_tyUSParam[1].iLaneID		            := p_tyRmtSetConfiguration.tyData.a_tyUpstreamConfigurations[p_udiRmtIndexUS2].iUpstreamLaneId;
			tyConfigurationWr.a_tyUSParam[1].sHostAddress           	:= p_tyRmtSetConfiguration.tyData.a_tyUpstreamConfigurations[p_udiRmtIndexUS2].sHostAddress;
			tyConfigurationWr.a_tyUSParam[1].uiHostPort	                := p_tyRmtSetConfiguration.tyData.a_tyUpstreamConfigurations[p_udiRmtIndexUS2].uiPort;
			tyConfigurationWr.a_tyUSParam[1].sUpstreamInterfaceId   	:= p_tyRmtSetConfiguration.tyData.a_tyUpstreamConfigurations[p_udiRmtIndexUS2].sUpstreamInterfaceId;
		END_IF

		IF p_bRmtFoundIndexUS3 THEN
			tyConfigurationWr.a_tyUSParam[2].iLaneID		            := p_tyRmtSetConfiguration.tyData.a_tyUpstreamConfigurations[p_udiRmtIndexUS3].iUpstreamLaneId;
			tyConfigurationWr.a_tyUSParam[2].sHostAddress           	:= p_tyRmtSetConfiguration.tyData.a_tyUpstreamConfigurations[p_udiRmtIndexUS3].sHostAddress;
			tyConfigurationWr.a_tyUSParam[2].uiHostPort	                := p_tyRmtSetConfiguration.tyData.a_tyUpstreamConfigurations[p_udiRmtIndexUS3].uiPort;
			tyConfigurationWr.a_tyUSParam[2].sUpstreamInterfaceId   	:= p_tyRmtSetConfiguration.tyData.a_tyUpstreamConfigurations[p_udiRmtIndexUS3].sUpstreamInterfaceId;
		END_IF

		IF p_bRmtFoundIndexUS4 THEN
			tyConfigurationWr.a_tyUSParam[3].iLaneID		            := p_tyRmtSetConfiguration.tyData.a_tyUpstreamConfigurations[p_udiRmtIndexUS4].iUpstreamLaneId;
			tyConfigurationWr.a_tyUSParam[3].sHostAddress           	:= p_tyRmtSetConfiguration.tyData.a_tyUpstreamConfigurations[p_udiRmtIndexUS4].sHostAddress;
			tyConfigurationWr.a_tyUSParam[3].uiHostPort	                := p_tyRmtSetConfiguration.tyData.a_tyUpstreamConfigurations[p_udiRmtIndexUS4].uiPort;
			tyConfigurationWr.a_tyUSParam[3].sUpstreamInterfaceId   	:= p_tyRmtSetConfiguration.tyData.a_tyUpstreamConfigurations[p_udiRmtIndexUS4].sUpstreamInterfaceId;
		END_IF

		IF p_bRmtFoundIndexDS1 THEN
			tyConfigurationWr.a_tyDSParam[0].iLaneID	            	:= p_tyRmtSetConfiguration.tyData.a_tyDownstreamConfigurations[p_udiRmtIndexDS1].iDownstreamLaneId;
			tyConfigurationWr.a_tyDSParam[0].uiSvrPort               	:= p_tyRmtSetConfiguration.tyData.a_tyDownstreamConfigurations[p_udiRmtIndexDS1].uiPort;
			tyConfigurationWr.a_tyDSParam[0].sDownstreamInterfaceId  	:= p_tyRmtSetConfiguration.tyData.a_tyDownstreamConfigurations[p_udiRmtIndexDS1].sDownstreamInterfaceId;
		END_IF

		IF p_bRmtFoundIndexDS2 THEN
			tyConfigurationWr.a_tyDSParam[1].iLaneID	            	:= p_tyRmtSetConfiguration.tyData.a_tyDownstreamConfigurations[p_udiRmtIndexDS2].iDownstreamLaneId;
			tyConfigurationWr.a_tyDSParam[1].uiSvrPort               	:= p_tyRmtSetConfiguration.tyData.a_tyDownstreamConfigurations[p_udiRmtIndexDS2].uiPort;
			tyConfigurationWr.a_tyDSParam[1].sDownstreamInterfaceId  	:= p_tyRmtSetConfiguration.tyData.a_tyDownstreamConfigurations[p_udiRmtIndexDS2].sDownstreamInterfaceId;
		END_IF

		IF p_bRmtFoundIndexDS3 THEN
			tyConfigurationWr.a_tyDSParam[2].iLaneID	            	:= p_tyRmtSetConfiguration.tyData.a_tyDownstreamConfigurations[p_udiRmtIndexDS3].iDownstreamLaneId;
			tyConfigurationWr.a_tyDSParam[2].uiSvrPort               	:= p_tyRmtSetConfiguration.tyData.a_tyDownstreamConfigurations[p_udiRmtIndexDS3].uiPort;
			tyConfigurationWr.a_tyDSParam[2].sDownstreamInterfaceId  	:= p_tyRmtSetConfiguration.tyData.a_tyDownstreamConfigurations[p_udiRmtIndexDS3].sDownstreamInterfaceId;
		END_IF

		IF p_bRmtFoundIndexDS4 THEN
			tyConfigurationWr.a_tyDSParam[3].iLaneID	            	:= p_tyRmtSetConfiguration.tyData.a_tyDownstreamConfigurations[p_udiRmtIndexDS4].iDownstreamLaneId;
			tyConfigurationWr.a_tyDSParam[3].uiSvrPort               	:= p_tyRmtSetConfiguration.tyData.a_tyDownstreamConfigurations[p_udiRmtIndexDS4].uiPort;
			tyConfigurationWr.a_tyDSParam[3].sDownstreamInterfaceId  	:= p_tyRmtSetConfiguration.tyData.a_tyDownstreamConfigurations[p_udiRmtIndexDS4].sDownstreamInterfaceId;
		END_IF

		IF p_tyRmtSetConfiguration.tyAvl.bMachineId = TRUE THEN

			tyConfigurationWr.a_tyUSParam[0].sMachineId		:= p_tyRmtSetConfiguration.tyData.sMachineId;
			tyConfigurationWr.a_tyDSParam[0].sMachineId		:= p_tyRmtSetConfiguration.tyData.sMachineId;
			tyConfigurationWr.tySvyParam.sMachineId		    := p_tyRmtSetConfiguration.tyData.sMachineId;

		END_IF

		IF p_tyRmtSetConfiguration.tyAvl.bSupervisorySystemPort = TRUE THEN

			tyConfigurationWr.tySvyParam.uiSvySvstemPort	:= p_tyRmtSetConfiguration.tyData.uiSupervisorySystemPort;

		END_IF

	ELSIF p_bUISaveHMIConfigure THEN //Save US, DS Configure in HMI

		tyConfigurationWr.a_tyUSParam[0]  := pa_tyUSParam[0]; //lane 1 US
		tyConfigurationWr.a_tyDSParam[0]  := pa_tyDSParam[0]; //lane 1 DS
		tyConfigurationWr.a_tyUSParam[1]  := pa_tyUSParam[1]; //lane 2 US
		tyConfigurationWr.a_tyDSParam[1]  := pa_tyDSParam[1]; //lane 2 DS
		tyConfigurationWr.a_tyUSParam[2]  := pa_tyUSParam[2]; //lane 3 US
		tyConfigurationWr.a_tyDSParam[2]  := pa_tyDSParam[2]; //lane 3 DS
		tyConfigurationWr.a_tyUSParam[3]  := pa_tyUSParam[3]; //lane 4 US
		tyConfigurationWr.a_tyDSParam[3]  := pa_tyDSParam[3]; //lane 4 DS

	ELSIF p_bUISaveHMISvyConfig THEN //Save Supervisory Configure in HMI

		tyConfigurationWr.tySvyParam  := p_tySvyParam;

	END_IF

END_ACTION
```

#### Act_Main.st - Do Not Change!!!
```iecst
(** 2021-08-01 **)
ACTION Act_Main:

	IF eStatOld <> eStat THEN
		fbDirCreate1(bEn := FALSE);
		fbDirCreate2(bEn := FALSE);
		fbDirCreate3(bEn := FALSE);
		fbDirCreate4(bEn := FALSE);
		fbFileRead1(bEn := FALSE);
		fbFileWrite1(bEn := FALSE);
		fbFileRead2(bEn := FALSE);
		fbFileWrite2(bEn := FALSE);
		fbFileRead3(bEn := FALSE);
		fbFileWrite3(bEn := FALSE);
		fbFileRead4(bEn := FALSE);
		fbFileWrite4(bEn := FALSE);
		fbFileRead5(bEn := FALSE);
		fbFileWrite5(bEn := FALSE);
		usiStep			:= 0;
		bFileNotFound	:= FALSE;

		sStatTxt	:= a_sStatText[eStat];

		eStatOld	:= eStat;

		eStatus		:= Busy;
	END_IF

	//Main
	CASE eStat OF

		HermesActIdle:
			eStatus	:= Idle;

		HermesActCreateDir:
			IF eStatus = Idle OR eStatus = Busy THEN

				eStatus	:= Busy;

				CASE usiStep OF
					0:
						fbDirCreate1(bEn := TRUE);
						IF fbDirCreate1.udiStatus = 0 THEN
							usiStep	:= 1;
						ELSIF fbDirCreate1.udiStatus < 65534 THEN
							eStatus		:= Error;

							IF fbDirCreate1.udiStatus = 1908 THEN
								udiStatus	:= 10000;	//Create User Directory Error
							ELSE
								udiStatus	:= fbDirCreate1.udiStatus;
							END_IF
						END_IF

					1:
						fbDirCreate2(bEn := TRUE);
						IF fbDirCreate2.udiStatus = 0 THEN
							usiStep	:= 2;
						ELSIF fbDirCreate2.udiStatus < 65534 THEN
							eStatus		:= Error;

							IF fbDirCreate2.udiStatus = 1908 THEN
								udiStatus	:= 10001;	//Create Retain Directory Error
							ELSE
								udiStatus	:= fbDirCreate2.udiStatus;
							END_IF
						END_IF

					2:
						fbDirCreate3(bEn := TRUE);
						IF fbDirCreate3.udiStatus = 0 THEN
							usiStep	:= 3;
						ELSIF fbDirCreate3.udiStatus < 65534 THEN
							eStatus		:= Error;

							IF fbDirCreate3.udiStatus = 1908 THEN
								udiStatus	:= 10010;	//Create Log Directory Error
							ELSE
								udiStatus	:= fbDirCreate3.udiStatus;
							END_IF
						END_IF

					3:
						fbDirCreate4(bEn := TRUE);
						IF fbDirCreate4.udiStatus = 0 THEN
							eStatus	:= Done;
						ELSIF fbDirCreate4.udiStatus < 65534 THEN
							eStatus		:= Error;

							IF fbDirCreate4.udiStatus = 1908 THEN
								udiStatus	:= 10011;	//Create Machine Parameter Directory Error
							ELSE
								udiStatus	:= fbDirCreate4.udiStatus;
							END_IF
						END_IF

				END_CASE

			END_IF

		HermesActReadRetainLane1:
			IF eStatus = Idle OR eStatus = Busy THEN

				eStatus	:= Busy;

				fbFileRead2.p_Dest	:= p_udiRetainDataAddr1;
				fbFileRead2.udiLen	:= p_udiRetainDataLen1;
				fbFileRead2(bEn := TRUE);

				IF fbFileRead2.udiStatus = 0 THEN
					eStatus	:= Done;
				ELSIF fbFileRead2.udiStatus < 65534 THEN
					eStatus	:= Error;

					IF fbFileRead2.udiStatus = 1900 THEN
						udiStatus	:= 10002;	//File Open Error While Reading Retain File
					ELSIF fbFileRead2.udiStatus = 1902 THEN
						udiStatus	:= 10003;	//File Read Error While Reading Retain File
					ELSIF fbFileRead2.udiStatus = 1904 THEN
						udiStatus	:= 10004;	//File Close Error While Reading Retain File
					ELSIF fbFileRead2.udiStatus = 1915 THEN
						eStatus			:= Done;
						bFileNotFound	:= TRUE;
					ELSE
						udiStatus	:= fbFileRead2.udiStatus;
					END_IF
				END_IF

			END_IF

		HermesActWriteRetainLane1:
			IF eStatus = Idle OR eStatus = Busy THEN

				eStatus	:= Busy;

				fbFileWrite2.p_Src	:= p_udiRetainDataAddr1;
				fbFileWrite2.udiLen	:= p_udiRetainDataLen1;
				fbFileWrite2(bEn := TRUE);

				IF fbFileWrite2.udiStatus = 0 THEN
					eStatus	:= Done;
				ELSIF fbFileWrite2.udiStatus < 65534 THEN
					eStatus	:= Error;

					IF fbFileWrite2.udiStatus = 1900 THEN
						udiStatus	:= 10005;	//File Open Error While Writing Retain File
					ELSIF fbFileWrite2.udiStatus = 1901 THEN
						udiStatus	:= 10006;	//File Create Error While Writing Retain File
					ELSIF fbFileWrite2.udiStatus = 1903 THEN
						udiStatus	:= 10007;	//File Write Error While Writing Retain File
					ELSIF fbFileWrite2.udiStatus = 1904 THEN
						udiStatus	:= 10008;	//File Close Error While Writing Retain File
					ELSIF fbFileWrite2.udiStatus = 1914 THEN
						udiStatus	:= 10009;	//Directory Does Not Exist While Writing Retain File
					ELSE
						udiStatus	:= fbFileWrite2.udiStatus;
					END_IF
				END_IF

			END_IF

		HermesActReadRetainLane2:
			IF eStatus = Idle OR eStatus = Busy THEN

				eStatus	:= Busy;

				fbFileRead3.p_Dest	:= p_udiRetainDataAddr2;
				fbFileRead3.udiLen	:= p_udiRetainDataLen2;
				fbFileRead3(bEn := TRUE);

				IF fbFileRead3.udiStatus = 0 THEN
					eStatus	:= Done;
				ELSIF fbFileRead3.udiStatus < 65534 THEN
					eStatus	:= Error;

					IF fbFileRead3.udiStatus = 1900 THEN
						udiStatus	:= 10032;	//File Open Error While Reading Retain File
					ELSIF fbFileRead3.udiStatus = 1902 THEN
						udiStatus	:= 10033;	//File Read Error While Reading Retain File
					ELSIF fbFileRead3.udiStatus = 1904 THEN
						udiStatus	:= 10034;	//File Close Error While Reading Retain File
					ELSIF fbFileRead3.udiStatus = 1915 THEN
						eStatus			:= Done;
						bFileNotFound	:= TRUE;
					ELSE
						udiStatus	:= fbFileRead3.udiStatus;
					END_IF
				END_IF

			END_IF

		HermesActWriteRetainLane2:
			IF eStatus = Idle OR eStatus = Busy THEN

				eStatus	:= Busy;

				fbFileWrite3.p_Src	:= p_udiRetainDataAddr2;
				fbFileWrite3.udiLen	:= p_udiRetainDataLen2;
				fbFileWrite3(bEn := TRUE);

				IF fbFileWrite3.udiStatus = 0 THEN
					eStatus	:= Done;
				ELSIF fbFileWrite3.udiStatus < 65534 THEN
					eStatus	:= Error;

					IF fbFileWrite3.udiStatus = 1900 THEN
						udiStatus	:= 10035;	//File Open Error While Writing Retain File
					ELSIF fbFileWrite3.udiStatus = 1901 THEN
						udiStatus	:= 10036;	//File Create Error While Writing Retain File
					ELSIF fbFileWrite3.udiStatus = 1903 THEN
						udiStatus	:= 10037;	//File Write Error While Writing Retain File
					ELSIF fbFileWrite3.udiStatus = 1904 THEN
						udiStatus	:= 10038;	//File Close Error While Writing Retain File
					ELSIF fbFileWrite3.udiStatus = 1914 THEN
						udiStatus	:= 10039;	//Directory Does Not Exist While Writing Retain File
					ELSE
						udiStatus	:= fbFileWrite3.udiStatus;
					END_IF
				END_IF

			END_IF

		HermesActReadRetainLane3:
			IF eStatus = Idle OR eStatus = Busy THEN

				eStatus	:= Busy;

				fbFileRead4.p_Dest	:= p_udiRetainDataAddr3;
				fbFileRead4.udiLen	:= p_udiRetainDataLen3;
				fbFileRead4(bEn := TRUE);

				IF fbFileRead4.udiStatus = 0 THEN
					eStatus	:= Done;
				ELSIF fbFileRead4.udiStatus < 65534 THEN
					eStatus	:= Error;

					IF fbFileRead4.udiStatus = 1900 THEN
						udiStatus	:= 10042;	//File Open Error While Reading Retain File
					ELSIF fbFileRead4.udiStatus = 1902 THEN
						udiStatus	:= 10043;	//File Read Error While Reading Retain File
					ELSIF fbFileRead4.udiStatus = 1904 THEN
						udiStatus	:= 10044;	//File Close Error While Reading Retain File
					ELSIF fbFileRead4.udiStatus = 1915 THEN
						eStatus			:= Done;
						bFileNotFound	:= TRUE;
					ELSE
						udiStatus	:= fbFileRead4.udiStatus;
					END_IF
				END_IF

			END_IF

		HermesActWriteRetainLane3:
			IF eStatus = Idle OR eStatus = Busy THEN

				eStatus	:= Busy;

				fbFileWrite4.p_Src	:= p_udiRetainDataAddr3;
				fbFileWrite4.udiLen	:= p_udiRetainDataLen3;
				fbFileWrite4(bEn := TRUE);

				IF fbFileWrite4.udiStatus = 0 THEN
					eStatus	:= Done;
				ELSIF fbFileWrite4.udiStatus < 65534 THEN
					eStatus	:= Error;

					IF fbFileWrite4.udiStatus = 1900 THEN
						udiStatus	:= 10045;	//File Open Error While Writing Retain File
					ELSIF fbFileWrite4.udiStatus = 1901 THEN
						udiStatus	:= 10046;	//File Create Error While Writing Retain File
					ELSIF fbFileWrite4.udiStatus = 1903 THEN
						udiStatus	:= 10047;	//File Write Error While Writing Retain File
					ELSIF fbFileWrite4.udiStatus = 1904 THEN
						udiStatus	:= 10048;	//File Close Error While Writing Retain File
					ELSIF fbFileWrite4.udiStatus = 1914 THEN
						udiStatus	:= 10049;	//Directory Does Not Exist While Writing Retain File
					ELSE
						udiStatus	:= fbFileWrite4.udiStatus;
					END_IF
				END_IF

			END_IF

		HermesActReadRetainLane4:
			IF eStatus = Idle OR eStatus = Busy THEN

				eStatus	:= Busy;

				fbFileRead5.p_Dest	:= p_udiRetainDataAddr4;
				fbFileRead5.udiLen	:= p_udiRetainDataLen4;
				fbFileRead5(bEn := TRUE);

				IF fbFileRead5.udiStatus = 0 THEN
					eStatus	:= Done;
				ELSIF fbFileRead5.udiStatus < 65534 THEN
					eStatus	:= Error;

					IF fbFileRead5.udiStatus = 1900 THEN
						udiStatus	:= 10052;	//File Open Error While Reading Retain File
					ELSIF fbFileRead5.udiStatus = 1902 THEN
						udiStatus	:= 10053;	//File Read Error While Reading Retain File
					ELSIF fbFileRead5.udiStatus = 1904 THEN
						udiStatus	:= 10054;	//File Close Error While Reading Retain File
					ELSIF fbFileRead5.udiStatus = 1915 THEN
						eStatus			:= Done;
						bFileNotFound	:= TRUE;
					ELSE
						udiStatus	:= fbFileRead5.udiStatus;
					END_IF
				END_IF

			END_IF

		HermesActWriteRetainLane4:
			IF eStatus = Idle OR eStatus = Busy THEN

				eStatus	:= Busy;

				fbFileWrite5.p_Src	:= p_udiRetainDataAddr4;
				fbFileWrite5.udiLen	:= p_udiRetainDataLen4;
				fbFileWrite5(bEn := TRUE);

				IF fbFileWrite5.udiStatus = 0 THEN
					eStatus	:= Done;
				ELSIF fbFileWrite5.udiStatus < 65534 THEN
					eStatus	:= Error;

					IF fbFileWrite5.udiStatus = 1900 THEN
						udiStatus	:= 10055;	//File Open Error While Writing Retain File
					ELSIF fbFileWrite5.udiStatus = 1901 THEN
						udiStatus	:= 10056;	//File Create Error While Writing Retain File
					ELSIF fbFileWrite5.udiStatus = 1903 THEN
						udiStatus	:= 10057;	//File Write Error While Writing Retain File
					ELSIF fbFileWrite5.udiStatus = 1904 THEN
						udiStatus	:= 10058;	//File Close Error While Writing Retain File
					ELSIF fbFileWrite5.udiStatus = 1914 THEN
						udiStatus	:= 10059;	//Directory Does Not Exist While Writing Retain File
					ELSE
						udiStatus	:= fbFileWrite5.udiStatus;
					END_IF
				END_IF

			END_IF

		HermesActReadConfig:
			IF eStatus = Idle OR eStatus = Busy THEN

				eStatus	:= Busy;

				fbFileRead1(bEn := TRUE);

				IF fbFileRead1.udiStatus = 0 THEN
					eStatus	:= Done;
					tyConfigurationWr := tyCurrConfiguration;
				ELSIF fbFileRead1.udiStatus < 65534 THEN
					eStatus	:= Error;

					IF fbFileRead1.udiStatus = 1900 THEN
						udiStatus	:= 10012;	//File Open Error While Reading Config File
					ELSIF fbFileRead1.udiStatus = 1902 THEN
						udiStatus	:= 10013;	//File Read Error While Reading Config File
					ELSIF fbFileRead1.udiStatus = 1904 THEN
						udiStatus	:= 10014;	//File Close Error While Reading Config File
					ELSIF fbFileRead1.udiStatus = 1915 THEN
						eStatus			:= Done;
						bFileNotFound	:= TRUE;
					ELSE
						udiStatus	:= fbFileRead1.udiStatus;
					END_IF
				END_IF

			END_IF

		HermesActWriteConfig:
			IF eStatus = Idle OR eStatus = Busy THEN

				eStatus	:= Busy;

				fbFileWrite1(bEn := TRUE);

				IF fbFileWrite1.udiStatus = 0 THEN
					eStatus	:= Done;
					tyCurrConfiguration := tyConfigurationWr;
				ELSIF fbFileWrite1.udiStatus < 65534 THEN
					eStatus	:= Error;

					IF fbFileWrite1.udiStatus = 1900 THEN
						udiStatus	:= 10015;	//File Open Error While Writing Config File
					ELSIF fbFileWrite1.udiStatus = 1901 THEN
						udiStatus	:= 10016;	//File Create Error While Writing Config File
					ELSIF fbFileWrite1.udiStatus = 1903 THEN
						udiStatus	:= 10017;	//File Write Error While Writing Config File
					ELSIF fbFileWrite1.udiStatus = 1904 THEN
						udiStatus	:= 10018;	//File Close Error While Writing Config File
					ELSIF fbFileWrite1.udiStatus = 1914 THEN
						udiStatus	:= 10019;	//Directory Does Not Exist While Writing Config File
					ELSE
						udiStatus	:= fbFileWrite1.udiStatus;
					END_IF
				END_IF

			END_IF

		ELSE
			IF eStatus = Idle OR eStatus = Busy THEN
				eStatus	:= Done;
			END_IF

	END_CASE

END_ACTION
```

#### Act_Alarm.st - Do Not Change!!!
```iecst
(** 2019-05-04 **)
ACTION Act_Alarm:

	//Error
	IF EDGEPOS(eStatus = Error) THEN

		tyAlmData.sProgNm		:= p_sProgNm;
		tyAlmData.udiCode		:= udiStatus;
		tyAlmData.eSeverity		:= AlmSeverityError;
		tyAlmData.udiRunTime	:= tyAlmData.udiRunTime + 1;
		tyAlmData.bAlm			:= TRUE;
		tyAlmData.udiModuleNum  := udiModuleNum;
		g_sHermesProgNm		:= p_sProgNm;
		//Get Error Message
		IF tyAlmData.udiCode < 10000 OR tyAlmData.udiCode > 10099 THEN
			tyAlmData.sAlmMsg	:= 'Unknown';
			tyAlmData.sRcyMsg	:= 'Unknown';
		ELSE
			tyAlmData.sAlmMsg	:= a_tyAlmText[tyAlmData.udiCode].sAlmText;
			tyAlmData.sRcyMsg	:= a_tyAlmText[tyAlmData.udiCode].sRcyText;
		END_IF

		sStatTxt	:= tyAlmData.sAlmMsg;

	ELSIF bRstErr AND (tyAlmData.udiCode <> 0) THEN

		tyAlmData.udiCode	:= 0;
		tyAlmData.eSeverity	:= AlmSeverityNA;
		tyAlmData.sAlmMsg	:= '';
		tyAlmData.sRcyMsg	:= '';
		tyAlmData.bAlm			:= FALSE;
		sStatTxt	:= a_sStatText[eStat];

	END_IF

END_ACTION
```

#### InputRef.var - Do Not Change!!!
```iecst
(*2019-05-04*)
(**)
(*General*)
VAR
	p_eAct : REFERENCE TO eHermesAction;
	p_udiRstErr : REFERENCE TO UDINT;
	p_bPrep : REFERENCE TO BOOL;
	p_bEn : REFERENCE TO BOOL;
	p_bDis : REFERENCE TO BOOL;
END_VAR
(**)
(*Configuration*)
(**)
(*Input*)
VAR
	pa_tyUSParam : REFERENCE TO ARRAY[0..c_diHermesConfigMaxIdx] OF tyHermesUSParam;
	pa_tyDSParam : REFERENCE TO ARRAY[0..c_diHermesConfigMaxIdx] OF tyHermesDSParam;
	p_tyRmtParam : REFERENCE TO tyHermesRmtParam;
	p_tySvyParam : REFERENCE TO tyHermesSvyParam;
	p_sMcId : REFERENCE TO STRING[30];
	p_bRmtHermesWriteConfig : REFERENCE TO BOOL;
	p_bSvyHermesWriteConfig : REFERENCE TO BOOL;
	p_bUISaveHMIConfigure : REFERENCE TO BOOL;
	p_bUISaveHMISvyConfig : REFERENCE TO BOOL;
	p_tyRmtSetConfiguration : REFERENCE TO tyHermesCurrentConfiguration;
	p_bRmtPrep : REFERENCE TO BOOL;
	p_bRmtEn : REFERENCE TO BOOL;
	p_tySvySetConfiguration : REFERENCE TO tyHermesCurrentConfiguration;
	p_bSvyPrep : REFERENCE TO BOOL;
	p_bSvyEn : REFERENCE TO BOOL;
	p_sRetainFileName1 : REFERENCE TO STRING[80];
	p_sRetainFileName2 : REFERENCE TO STRING[80];
	p_sRetainFileName3 : REFERENCE TO STRING[80];
	p_sRetainFileName4 : REFERENCE TO STRING[80];
	p_udiRetainDataAddr1 : REFERENCE TO UDINT;
	p_udiRetainDataLen1 : REFERENCE TO UDINT;
	p_udiRetainDataAddr2 : REFERENCE TO UDINT;
	p_udiRetainDataLen2 : REFERENCE TO UDINT;
	p_udiRetainDataAddr3 : REFERENCE TO UDINT;
	p_udiRetainDataLen3 : REFERENCE TO UDINT;
	p_udiRetainDataAddr4 : REFERENCE TO UDINT;
	p_udiRetainDataLen4 : REFERENCE TO UDINT;
	p_sConfigFileName : REFERENCE TO STRING[80];
	p_sProgNm : REFERENCE TO STRING[15];
	p_bNtSettingsLoadDone : REFERENCE TO BOOL;
END_VAR
(**)
(*RmtHermes*)
VAR
	p_bRmtFoundIndexUS1 : REFERENCE TO BOOL;
	p_bRmtFoundIndexUS2 : REFERENCE TO BOOL;
	p_bRmtFoundIndexUS3 : REFERENCE TO BOOL;
	p_bRmtFoundIndexUS4 : REFERENCE TO BOOL;
	p_bRmtFoundIndexDS1 : REFERENCE TO BOOL;
	p_bRmtFoundIndexDS2 : REFERENCE TO BOOL;
	p_bRmtFoundIndexDS3 : REFERENCE TO BOOL;
	p_bRmtFoundIndexDS4 : REFERENCE TO BOOL;
	p_udiRmtIndexUS1 : REFERENCE TO UDINT;
	p_udiRmtIndexUS2 : REFERENCE TO UDINT;
	p_udiRmtIndexUS3 : REFERENCE TO UDINT;
	p_udiRmtIndexUS4 : REFERENCE TO UDINT;
	p_udiRmtIndexDS1 : REFERENCE TO UDINT;
	p_udiRmtIndexDS2 : REFERENCE TO UDINT;
	p_udiRmtIndexDS3 : REFERENCE TO UDINT;
	p_udiRmtIndexDS4 : REFERENCE TO UDINT;
END_VAR
(**)
(*SvyHermes*)
VAR
	p_bSvyFoundIndexUS1 : REFERENCE TO BOOL;
	p_bSvyFoundIndexUS2 : REFERENCE TO BOOL;
	p_bSvyFoundIndexUS3 : REFERENCE TO BOOL;
	p_bSvyFoundIndexUS4 : REFERENCE TO BOOL;
	p_bSvyFoundIndexDS1 : REFERENCE TO BOOL;
	p_bSvyFoundIndexDS2 : REFERENCE TO BOOL;
	p_bSvyFoundIndexDS3 : REFERENCE TO BOOL;
	p_bSvyFoundIndexDS4 : REFERENCE TO BOOL;
	p_udiSvyIndexUS1 : REFERENCE TO UDINT;
	p_udiSvyIndexUS2 : REFERENCE TO UDINT;
	p_udiSvyIndexUS3 : REFERENCE TO UDINT;
	p_udiSvyIndexUS4 : REFERENCE TO UDINT;
	p_udiSvyIndexDS1 : REFERENCE TO UDINT;
	p_udiSvyIndexDS2 : REFERENCE TO UDINT;
	p_udiSvyIndexDS3 : REFERENCE TO UDINT;
	p_udiSvyIndexDS4 : REFERENCE TO UDINT;
END_VAR
(**)
```

#### Local.var - Do Not Change!!!
```iecst
(*2021-08-01*)
(**)
(*Local Action, State & Status*)
VAR
	eAct : eHermesAction := HermesActIdle;
	eStat : eHermesAction := HermesActIdle;
	eStatus : eFBStatus := Idle;
	udiStatus : UDINT := 0;
	sStatTxt : STRING[200] := '';
	a_sStatText : ARRAY[0..50] OF STRING[200] := ['Idling','Background Starting Operations','Background Stopping Operations','Deleting Old Log File','Creating Directory','Writing Retain File','Reading Retain File','Writing Configuration File','Reading Configuration File',42('')];
END_VAR
(**)
(*Local Alarm*)
VAR
	tyAlmData : tyAlmDat;
	a_tyAlmText : ARRAY[10000..10099] OF tyAlmTxt := [(sAlmText:='Create User Directory Error',sRcyText:='An Error Occurred While Attempting To Create User Directory. Please Contact Nutek For A Possible Solution'),(sAlmText:='Create Retain Directory Error',sRcyText:='An Error Occurred While Attempting To Create Retain Directory. Please Contact Nutek For A Possible Solution'),(sAlmText:='File Open Error While Reading Retain File',sRcyText:='An Error Was Encountered While Trying To Open File. Please Contact Nutek For A Possible Solution.'),(sAlmText:='File Read Error While Reading Retain File',sRcyText:='An Error Was Encountered While Trying To Read File. Please Contact Nutek For A Possible Solution.'),(sAlmText:='File Close Error While Reading Retain File',sRcyText:='An Error Was Encountered While Trying To Close File. Please Contact Nutek For A Possible Solution.'),(sAlmText:='File Open Error While Writing Retain File',sRcyText:='An Error Was Encountered While Trying To Open File. Please Contact Nutek For A Possible Solution.'),(sAlmText:='File Create Error While Writing Retain File',sRcyText:='An Error Was Encountered While Trying To Create File. Please Contact Nutek For A Possible Solution.'),(sAlmText:='File Write Error While Writing Retain File',sRcyText:='An Error Was Encountered While Trying To Write File. Please Contact Nutek For A Possible Solution.'),(sAlmText:='File Close Error While Writing Retain File',sRcyText:='An Error Was Encountered While Trying To Close File. Please Contact Nutek For A Possible Solution.'),(sAlmText:='Directory Does Not Exist While Writing Retain File',sRcyText:='The Directory Does Not Exist. Please Contact Nutek For A Possible Solution.'),(sAlmText:='Create Log Directory Error',sRcyText:='An Error Occurred While Attempting To Create Log Directory. Please Contact Nutek For A Possible Solution'),(sAlmText:='Create Machine Parameter Directory Error',sRcyText:='An Error Occurred While Attempting To Create Machine Parameter Directory. Please Contact Nutek For A Possible Solution'),(sAlmText:='File Open Error While Reading Config File',sRcyText:='An Error Was Encountered While Trying To Open File. Please Contact Nutek For A Possible Solution.'),(sAlmText:='File Read Error While Reading Config File',sRcyText:='An Error Was Encountered While Trying To Read File. Please Contact Nutek For A Possible Solution.'),(sAlmText:='File Close Error While Reading Config File',sRcyText:='An Error Was Encountered While Trying To Close File. Please Contact Nutek For A Possible Solution.'),(sAlmText:='File Open Error While Writing Config File',sRcyText:='An Error Was Encountered While Trying To Open File. Please Contact Nutek For A Possible Solution.'),(sAlmText:='File Create Error While Writing Config File',sRcyText:='An Error Was Encountered While Trying To Create File. Please Contact Nutek For A Possible Solution.'),(sAlmText:='File Write Error While Writing Config File',sRcyText:='An Error Was Encountered While Trying To Write File. Please Contact Nutek For A Possible Solution.'),(sAlmText:='File Close Error While Writing Config File',sRcyText:='An Error Was Encountered While Trying To Close File. Please Contact Nutek For A Possible Solution.'),(sAlmText:='Directory Does Not Exist While Writing Config File',sRcyText:='The Directory Does Not Exist. Please Contact Nutek For A Possible Solution.'),(0),2(0),3((0)),0,3((0)),(sAlmText:='File Open Error While Writing Retain File Lane 2',sRcyText:='An Error Was Encountered While Trying To Open File. Please Contact Nutek For A Possible Solution.'),(0),(sAlmText:='File Open Error While Reading Lane 2 Retain File',sRcyText:='An Error Was Encountered While Trying To Open File. Please Contact Nutek For A Possible Solution.'),(sAlmText:='File Read Error While Reading Lane 2 Retain File',sRcyText:='An Error Was Encountered While Trying To Read File. Please Contact Nutek For A Possible Solution.'),(sAlmText:='File Close Error While Reading Lane 2 Retain File',sRcyText:='An Error Was Encountered While Trying To Close File. Please Contact Nutek For A Possible Solution.'),(sAlmText:='File Open Error While Writing Lane 2 Retain File',sRcyText:='An Error Was Encountered While Trying To Open File. Please Contact Nutek For A Possible Solution.'),(sAlmText:='File Create Error While Writing Lane 2 Retain File',sRcyText:='An Error Was Encountered While Trying To Create File. Please Contact Nutek For A Possible Solution.'),(sAlmText:='File Write Error While Writing Lane 2 Retain File',sRcyText:='An Error Was Encountered While Trying To Write File. Please Contact Nutek For A Possible Solution.'),(sAlmText:='File Close Error While Writing Lane 2 Retain File',sRcyText:='An Error Was Encountered While Trying To Close File. Please Contact Nutek For A Possible Solution.'),(sAlmText:='Directory Does Not Exist While Writing Lane 2 Retain File',sRcyText:='The Directory Does Not Exist. Please Contact Nutek For A Possible Solution.'),2((0)),(sAlmText:='File Open Error While Reading Lane 3 Retain File',sRcyText:='An Error Was Encountered While Trying To Open File. Please Contact Nutek For A Possible Solution.'),(sAlmText:='File Read Error While Reading Lane 3 Retain File',sRcyText:='An Error Was Encountered While Trying To Read File. Please Contact Nutek For A Possible Solution.'),(sAlmText:='File Close Error While Reading Lane 3 Retain File',sRcyText:='An Error Was Encountered While Trying To Close File. Please Contact Nutek For A Possible Solution.'),(sAlmText:='File Open Error While Writing Lane 3 Retain File',sRcyText:='An Error Was Encountered While Trying To Open File. Please Contact Nutek For A Possible Solution.'),(sAlmText:='File Create Error While Writing Lane 3 Retain File',sRcyText:='An Error Was Encountered While Trying To Create File. Please Contact Nutek For A Possible Solution.'),(sAlmText:='File Write Error While Writing Lane 3 Retain File',sRcyText:='An Error Was Encountered While Trying To Write File. Please Contact Nutek For A Possible Solution.'),(sAlmText:='File Close Error While Writing Lane 3 Retain File',sRcyText:='An Error Was Encountered While Trying To Close File. Please Contact Nutek For A Possible Solution.'),(sAlmText:='Directory Does Not Exist While Writing Lane 3 Retain File',sRcyText:='The Directory Does Not Exist. Please Contact Nutek For A Possible Solution.'),2((0)),(sAlmText:='File Open Error While Reading Lane 4 Retain File',sRcyText:='An Error Was Encountered While Trying To Open File. Please Contact Nutek For A Possible Solution.'),(sAlmText:='File Read Error While Reading Lane 4 Retain File',sRcyText:='An Error Was Encountered While Trying To Read File. Please Contact Nutek For A Possible Solution.'),(sAlmText:='File Close Error While Reading Lane 4 Retain File',sRcyText:='An Error Was Encountered While Trying To Close File. Please Contact Nutek For A Possible Solution.'),(sAlmText:='File Open Error While Writing Lane 4 Retain File',sRcyText:='An Error Was Encountered While Trying To Open File. Please Contact Nutek For A Possible Solution.'),(sAlmText:='File Create Error While Writing Lane 4 Retain File',sRcyText:='An Error Was Encountered While Trying To Create File. Please Contact Nutek For A Possible Solution.'),(sAlmText:='File Write Error While Writing Lane 4 Retain File',sRcyText:='An Error Was Encountered While Trying To Write File. Please Contact Nutek For A Possible Solution.'),(sAlmText:='File Close Error While Writing Lane 4 Retain File',sRcyText:='An Error Was Encountered While Trying To Close File. Please Contact Nutek For A Possible Solution.'),(sAlmText:='Directory Does Not Exist While Writing Lane 4 Retain File',sRcyText:='The Directory Does Not Exist. Please Contact Nutek For A Possible Solution.'),40((0))];
END_VAR
(**)
(*Local Output*)
VAR
	bFileNotFound : BOOL;
	tyCurrConfiguration : tyHermesConfiguration := (a_tyUSParam:=[(tSndAlive:=T#60s,iLaneID:=1,sHostAddress:='127.0.0.1',uiHostPort:=501),3(0)],a_tyDSParam:=[(tSndAlive:=T#60s,uiSvrPort:=502,iLaneID:=1),3((0))]);
	tyConfigurationWr : tyHermesConfiguration;
END_VAR
(**)
(*Local Input*)
VAR
	udiRstErr : UDINT := 0;
	bPrep : BOOL := TRUE;
	bEn : BOOL := TRUE;
	bDis : BOOL := FALSE;
	a_tyUSParam : ARRAY[0..c_diHermesConfigMaxIdx] OF tyHermesUSParam;
	a_tyDSParam : ARRAY[0..c_diHermesConfigMaxIdx] OF tyHermesDSParam;
	tyRmtParam : tyHermesRmtParam;
	tySvyParam : tyHermesSvyParam;
	tyRmtSetConfiguration : tyHermesCurrentConfiguration;
	tySvySetConfiguration : tyHermesCurrentConfiguration;
	bRmtPrep : BOOL := FALSE;
	bRmtEn : BOOL := FALSE;
	bSvyPrep : BOOL := FALSE;
	bSvyEn : BOOL := FALSE;
	sRetainFileName1 : STRING[80] := 'HermesLane1.dat';
	sRetainFileName2 : STRING[80] := 'HermesLane2.dat';
	sRetainFileName3 : STRING[80] := 'HermesLane3.dat';
	sRetainFileName4 : STRING[80] := 'HermesLane4.dat';
	udiRetainDataAddr1 : UDINT;
	udiRetainDataLen1 : UDINT;
	udiRetainDataAddr2 : UDINT;
	udiRetainDataLen2 : UDINT;
	udiRetainDataAddr3 : UDINT;
	udiRetainDataLen3 : UDINT;
	udiRetainDataAddr4 : UDINT;
	udiRetainDataLen4 : UDINT;
	sConfigFileName : STRING[80] := 'Hermes.dat';
	sProgNm : STRING[15] := 'Hermes';
	bNtSettingsLoadDone : BOOL := TRUE;
	bRmtHermesWriteConfig : BOOL := TRUE;
	bSvyHermesWriteConfig : BOOL := TRUE;
	bUISaveHMIConfigure : BOOL := TRUE;
	bUISaveHMISvyConfig : BOOL := TRUE;
	sMcId : STRING[30] := '';
	bRmtFoundIndexUS1 : BOOL := FALSE;
	bRmtFoundIndexUS2 : BOOL := FALSE;
	bRmtFoundIndexUS3 : BOOL := FALSE;
	bRmtFoundIndexUS4 : BOOL := FALSE;
	bRmtFoundIndexDS1 : BOOL := FALSE;
	bRmtFoundIndexDS2 : BOOL := FALSE;
	bRmtFoundIndexDS3 : BOOL := FALSE;
	bRmtFoundIndexDS4 : BOOL := FALSE;
	udiRmtIndexUS1 : UDINT := 0;
	udiRmtIndexUS2 : UDINT := 0;
	udiRmtIndexUS3 : UDINT := 0;
	udiRmtIndexUS4 : UDINT := 0;
	udiRmtIndexDS1 : UDINT := 0;
	udiRmtIndexDS2 : UDINT := 0;
	udiRmtIndexDS3 : UDINT := 0;
	udiRmtIndexDS4 : UDINT := 0;
	bSvyFoundIndexUS1 : BOOL := FALSE;
	bSvyFoundIndexUS2 : BOOL := FALSE;
	bSvyFoundIndexUS3 : BOOL := FALSE;
	bSvyFoundIndexUS4 : BOOL := FALSE;
	bSvyFoundIndexDS1 : BOOL := FALSE;
	bSvyFoundIndexDS2 : BOOL := FALSE;
	bSvyFoundIndexDS3 : BOOL := FALSE;
	bSvyFoundIndexDS4 : BOOL := FALSE;
	udiSvyIndexUS1 : UDINT := 0;
	udiSvyIndexUS2 : UDINT := 0;
	udiSvyIndexUS3 : UDINT := 0;
	udiSvyIndexUS4 : UDINT := 0;
	udiSvyIndexDS1 : UDINT := 0;
	udiSvyIndexDS2 : UDINT := 0;
	udiSvyIndexDS3 : UDINT := 0;
	udiSvyIndexDS4 : UDINT := 0;
END_VAR
(**)
(*Local*)
VAR
	bRstErr : BOOL;
	udiRstErrOld : UDINT;
	bInitDone : BOOL;
	bInitialDone : BOOL;
	bHermesWriteRetain : BOOL;
	bHermesWriteRetainLane1 : BOOL;
	bHermesWriteRetainLane2 : BOOL;
	bHermesWriteRetainLane3 : BOOL;
	bHermesWriteRetainLane4 : BOOL;
	usiStep : USINT;
	tyConfigurationHMI : tyHermesConfiguration;
	eStatOld : eHermesAction := HermesActIdle;
	fbDirCreate1 : fbDirCreate;
	fbDirCreate2 : fbDirCreate;
	fbDirCreate3 : fbDirCreate;
	fbDirCreate4 : fbDirCreate;
	fbFileRead1 : fbFileFullRead;
	fbFileWrite1 : fbFileFullWrite;
	fbFileRead2 : fbFileFullRead;
	fbFileWrite2 : fbFileFullWrite;
	fbFileRead3 : fbFileFullRead;
	fbFileWrite3 : fbFileFullWrite;
	fbFileRead4 : fbFileFullRead;
	fbFileWrite4 : fbFileFullWrite;
	fbFileRead5 : fbFileFullRead;
	fbFileWrite5 : fbFileFullWrite;
	i : INT;
	bVoid : BOOL;
	udiModuleNum : UDINT := 2901;
END_VAR
```

### USHermesA.var - Change By Project
```iecst
(*2019-06-10*)
(**)
(*Action & State & Status*)
VAR
	p_USHermesAStat : UDINT;
	p_USHermesAStatus : UDINT;
	p_USHermesAStatTxt : UDINT;
END_VAR
(**)
(*Alarm*)
VAR
	p_USHermesAAlmData : UDINT;
	p_USHermesAAlmData1 : UDINT;
	p_USHermesAAlmData2 : UDINT;
	p_USHermesAAlmData3 : UDINT;
	p_USHermesAAlmData4 : UDINT;
	p_USHermesAAlmData5 : UDINT;
	p_USHermesAInfoData : UDINT;
	p_USHermesAInfoData1 : UDINT;
	p_USHermesAInfoData2 : UDINT;
END_VAR
(**)
(*Output*)
VAR
	p_USHermesATableDataBrdAvl : UDINT;
	p_USHermesATableDataBrdAvlTtlIdx : UDINT;
	p_USHermesAConnected : UDINT;
	p_USHermesAHandshakeDone : UDINT;
	p_USHermesAAccDataReq : UDINT;
	p_USHermesABFAccDataReq : UDINT;
	p_USHermesAOverWriteSlt : UDINT;
	p_USHermesAOverWriteWidth : UDINT;
	p_USHermesAReqRecipeNm : UDINT;
	p_USHermesAReqWidthInUM : UDINT;
	p_USHermesAReqMinSltValue : UDINT;
	p_USHermesAReqMaxSltValue : UDINT;
	p_USHermesAReqPitch : UDINT;
	p_USHermesAUSRdy : UDINT;
	p_USHermesADSRdy : UDINT;
	p_USHermesAUSGdRdy : UDINT;
	p_USHermesADSGdRdy : UDINT;
	p_USHermesATransporting : UDINT;
	p_USHermesAStopTransport : UDINT;
	p_USHermesABlkUS : UDINT;
	p_USHermesAInternalSnd : UDINT;
	p_USHermesAAccDataMnl : UDINT;
	p_USHermesAStopTransportSnd : UDINT;
	p_USHermesABoardArrivedData : UDINT;
	p_USHermesARcvBoardInfoOk : UDINT;
	p_USHermesARcvbBoardInfoIncompl : UDINT;
	p_USHermesABoardInfoData : UDINT;
	p_USHermesANextAvlPCBTimer : UDINT;
	p_USHermesAManuallInsertLastZone : UDINT;
	p_USHermesABoardAvailableRcv : UDINT;
	p_USHermesABoardForecastRcv : UDINT;
END_VAR
(*//changed*)
VAR
	p_USHermesABAAccepted : UDINT;
	p_USHermesABFAccepted : UDINT;
	p_USHermesATopBtmBarcode : UDINT;
END_VAR
```

### Program Logical/Hermes/USHermesA (IEC) - 1.00.0 - NtHermes v5.00.0 , NtTCP v5.00.0 , NtMessage v5.00.0

#### InputRef.var
```iecst
(*2021-08-01*)
(**)
(*General*)
VAR
	p_eAct : REFERENCE TO eHermesAction;
	p_udiRstErr : REFERENCE TO UDINT;
	p_bPrep : REFERENCE TO BOOL;
	p_bEn : REFERENCE TO BOOL;
	p_bDis : REFERENCE TO BOOL;
END_VAR
(**)
(*Configuration*)
VAR
	p_tyParam : REFERENCE TO tyHermesUSParam;
	p_sIPAddr : REFERENCE TO STRING[15];
	p_tyDTStructure : REFERENCE TO DTStructure;
	p_dtCurrDT : REFERENCE TO DATE_AND_TIME;
	p_sMcId : REFERENCE TO STRING[80];
END_VAR
(**)
(*Input*)
VAR
	p_bRdyRcv : REFERENCE TO BOOL;
	p_bRdyTransport : REFERENCE TO BOOL;
	p_bRcvCompl : REFERENCE TO BOOL;
	p_bRcvIncompl : REFERENCE TO BOOL;
	p_bRcvNotStart : REFERENCE TO BOOL;
	p_bBAWidthEn : REFERENCE TO BOOL; (*Board Available Check Width*)
	p_bBASltEn : REFERENCE TO BOOL; (*Board Available Check Slot*)
	p_bBFWidthEn : REFERENCE TO BOOL; (*Board Forecast Check Width*)
	p_bBFSltEn : REFERENCE TO BOOL; (*Board Forecast Check Slot*)
	p_sRecipeNm : REFERENCE TO STRING[254];
	p_sInterfaceId : REFERENCE TO STRING[80];
	p_sVersion : REFERENCE TO STRING[7];
	p_eFailedBoard : REFERENCE TO eHermesFailedBoard;
	p_diWidthInUM : REFERENCE TO DINT;
	p_diMinSltValue : REFERENCE TO DINT;
	p_diMaxSltValue : REFERENCE TO DINT;
	p_diPitch : REFERENCE TO DINT;
	p_diTtlSlt : REFERENCE TO DINT;
	p_diSltToSltInUM : REFERENCE TO DINT;
	p_udiSndBffrSize : REFERENCE TO UDINT;
	p_udiRcvBffrSize : REFERENCE TO UDINT;
	p_udiAliveIdleTimeInSec : REFERENCE TO UDINT;
	p_tConnTimeOut : REFERENCE TO TIME;
	p_diTransferInTO : REFERENCE TO DINT;
	p_bOpsRun : REFERENCE TO BOOL;
	p_bInterruptSen : REFERENCE TO BOOL;
	p_udiFileKeepDay : REFERENCE TO UDINT;
	p_sProgNm : REFERENCE TO STRING[15];
	p_bNtSettingsLoadDone : REFERENCE TO BOOL;
	p_bAccDataRdy : REFERENCE TO BOOL;
	p_bRmtPrep : REFERENCE TO BOOL;
	p_bRmtEn : REFERENCE TO BOOL;
	p_bSvyPrep : REFERENCE TO BOOL;
	p_bSvyEn : REFERENCE TO BOOL;
	p_bAccNewRcpCond : REFERENCE TO BOOL;
	p_sInfoMsg : REFERENCE TO STRING[200];
	p_sInfoMsg1 : REFERENCE TO STRING[200];
	p_sInfoMsg2 : REFERENCE TO STRING[200];
	pa_tyProdRcpList : REFERENCE TO ARRAY[1..c_udiProdRcpMax] OF tyProdRcpParam;
	p_tyProdRcpCurrRcp : REFERENCE TO tyProdRcpParam;
	p_bMcParamMnlAccData : REFERENCE TO BOOL;
	p_bOpsGConv1HvBrd : REFERENCE TO BOOL;
	p_bManualInsertZoneHvBrd : REFERENCE TO BOOL;
	p_bUIAccData : REFERENCE TO BOOL;
	p_bQueryBoardInfo : REFERENCE TO BOOL;
	p_sTopBarcode : REFERENCE TO STRING[254];
	p_sBottomBarcode : REFERENCE TO STRING[254];
	p_tyHermesConfiguration : REFERENCE TO tyHermesConfiguration;
	p_bTransportFinished : REFERENCE TO BOOL;
	p_bManualInsertEndSen : REFERENCE TO BOOL;
	p_bInternalUse : REFERENCE TO BOOL;
	p_sInternalRcv : REFERENCE TO STRING[65535];
	p_usiLinkProdRcpCurrRcpMcMod : REFERENCE TO USINT;
	p_bNewIncomingBoard : REFERENCE TO BOOL;
	p_bQueryBypassWorkOrder : REFERENCE TO BOOL;
	p_bSiemensMcModeChgPrep : REFERENCE TO BOOL;
	p_bNtParamAutoRcpPrep : REFERENCE TO BOOL;
	p_bMcParamAutoRcpDis : REFERENCE TO BOOL;
	p_eNtParamAutoRcpPrecededBy : REFERENCE TO eAutoRcpPreceded;
END_VAR
```

#### InputRef_Link.var
```iecst
(*2019-06-28*)
(**)
VAR
	p_bLinkStartupRun : REFERENCE TO BOOL;
	p_eLinkMcParamUSCommMod : REFERENCE TO eMcSetCommMod;
	bHermesRun : BOOL;
	bHermesStop : BOOL;
END_VAR
(**)
VAR
	p_bLinkDILeftSen : REFERENCE TO BOOL;
	p_eLinkTravLifULPosGo : REFERENCE TO eTravLifULPos;
	p_bLinkOpsTravLifULUSComm : REFERENCE TO BOOL;
END_VAR
(**)
VAR
	sWidthInUMTemp : STRING[80];
END_VAR
```
